FUNCTION_BLOCK FB_BMS
VAR PERSISTENT
	ui_CycleCount				: UINT;
	r_CumDischargeEnergy		: REAL; // kWh
	r_CumChargeEnergy			: REAL; // kWh
	r_maxVoltageEver	 		: REAL;
	r_maxChargeCurrentEver		: REAL;
	r_maxDischargeCurrentEver	: REAL;
	dt_LastCalibrationDate		: DT;
END_VAR

VAR_IN_OUT CONSTANT
	st_params	: st_BMS_Params;
END_VAR

VAR_IN_OUT
 	st_service	: st_BMS_service;
END_VAR

VAR_OUTPUT
	PowerStatus: eHVDC_Powerstatus := 0;
END_VAR
VAR_INPUT
	Set 					: st_BMS_Set;
	b_HVDCEnable			: BOOL;
	by_NoOfStrings			: BYTE;
END_VAR

VAR_OUTPUT
	get						: st_BMS_Get;
	b_InternalHVDCAllowed	:	BOOL;
END_VAR

VAR	
	InitDone			:	Bool := false;
	b_HVDC_OnRq			: BOOL;	
	FBState					:	ePOUState;
	IO					:	FB_BMS_IO;
	InitTimeout			: 	TON := (PT:=T#3S);
	BMS_24V_StartupTimer : TON := (PT := TIME#2S0MS);
	
	DeviceIDcounter		: WORD;
	
	//SFC
	SFCInit				: BOOL := FALSE;
	SFCReset			: BOOL := FALSE;
	
	//Modbus
	b_MBComErrorActive	: 	BOOL 	:= FALSE;
	ComTimer			:	Ton := (PT := TIME#100MS);
	t_TimeOut			: 	TIME := T#500MS;
	
	ResetBMS	:	Bool; 
	b_BMSShutdownRequested: BOOL;
	
	BMSReadIntervalTimer	 : TON := (PT := TIME#1S0MS);
	
	b_ManualReset	:BOOL;
	BMSDataValid		:	Bool;
	
	arDatalogMBMU	: ARRAY [0..58] OF WORD;
	arDatalogSBMU	: ARRAY[0..3] OF ARRAY[0..55] OF WORD;
	ARDatalogEMS	: ARRAY [0..16] OF WORD;
	
	AutoSOCCalibrationRequired	:	Bool;
END_VAR

VAR CONSTANT
	e_ID 				: eObject_ID := eObject_ID.Battery;
END_VAR

BMSDatalogger(b_enable := InitDone);
(*
FB_BMS

Inputs
	Set.b_EnableBMS				:	BOOL;
		Start BMS SFC sequence and initializes BMS. False means full BMS powerdown, so no status logging.
		With HVDC enabled, setting this value to False has no effect. Only after HVDC powerdown this value is tested.
		
	Set.b_ClearFault				:	BOOL;
		Clear errors and warning in BMS system. Set to true to initiate reset. Value resets automatically to false.
	
	Set.b_HVDC_Required			: 	BOOL;
		Set by FB_internalPowersupply. True initiates and keeps HVDC on, False initiates and retains powerdown

Outputs
	BMSGET
		-Some general status info
		-BATTinfo	struct with main operation battery data
		-MBMU_Status 	struct with detailed MBMU data
		-SBMU			Struct with detailed data per SBMU
		-Events			Warnings & Errors as per Sunspec list.
*)

IF InitDone THEN
	//INIT step
	//b_MBComErrorActive := FALSE;
	
	//CALL methods/functions
	//Link MBMU data when appropriate
	GetBatteryInfo(in := get.MBMU.BatteryStatus, OUT:= get.BatteryInfo);
	
	IF st_params.b_EnableAutoCalibration THEN
		IF dt_LastCalibrationDate > gvl.dt_SystemDateTime OR 
			(dt_LastCalibrationDate + st_params.T_AutoCalibrationInterval) < gvl.dt_SystemDateTime THEN
			get.T_RemainingTimeToAutoCalibration := T#0S;
			AutoSOCCalibrationRequired := TRUE;
		ELSE
			AutoSOCCalibrationRequired := FALSE;
			get.T_RemainingTimeToAutoCalibration := (dt_LastCalibrationDate + st_params.T_AutoCalibrationInterval) - gvl.dt_SystemDateTime;
		END_IF
	ELSE
		AutoSOCCalibrationRequired := FALSE;
		get.T_RemainingTimeToAutoCalibration := ST_Params.t_AutoCalibrationInterval;
	END_IF

		
	

	//get.LastCalibrationTime := dt_LastCalibrationDate;
	
	IF get.BatteryInfo.r_SOC < st_params.r_InternalConditioningSoCMin OR get.BatteryInfo.ar_CellVoltage[eSubValues.Minimum] < 3 THEN
		b_InternalHVDCAllowed := FALSE;
	ELSE
		b_InternalHVDCAllowed := TRUE;
	END_IF
	
	IO();
	
	BMSReadIntervalTimer(in:= not BMSReadIntervalTimer.Q);
	
	//Reset ErrorActive before entering SFC. 
	//any remaining error in the Modbus methods will set Erroractive again. 
	//This is pushed to events in BMS_Diagnostics
	
	//TEMPBMSHB();
	//hv required not allowed if BMS not enabled
	IF set.b_enable AND FBstate <> epoustate.EMSTOP THEN
		b_HVDC_OnRq := b_HVDCEnable OR st_params.b_forcePrecharging;
		
	ELSE
		b_HVDC_OnRq := FALSE;	
	END_IF
	
	//shutdown allowed if hvdc is offline
	b_BMSShutdownRequested := (NOT Set.b_Enable) AND get.MBMU.BatteryStatus.e_BMS_PowerOnStatus <> ePowerOnStatus.On; 
	
	IF b_ManualReset THEN
		Reset();
	END_IF
	
	//SFC delayed pulse trigger
	BMSSFC();
	
	BMS_Diagnostics();
	
	BMSDataValid := ((NOT get.Events.b_COMMUNICATION_ERROR) AND NOT (get.BatteryInfo.e_BMS_Status = eBMS_Status.Init));
END_IF

ACTION aBMSPoweroff:
IO.b_BMSEnable := FALSE;

get.BatteryInfo.b_BMSHeartBeatOK := FALSE;
get.BatteryInfo.e_BMS_PowerOnStatus := ePowerOnStatus.Off;
get.BatteryInfo.e_BMS_Status := eBMS_Status.Off;

get.MBMU.BatteryStatus.b_BMSHeartBeatOK := FALSE;
get.MBMU.BatteryStatus.e_BMS_PowerOnStatus := ePowerOnStatus.Off;
get.MBMU.BatteryStatus.e_BMS_Status := eBMS_Status.Off;

FBState := ePOUState.OFF;
END_ACTION

ACTION aBMSPowerOn:

//230V inverter requires some startup time. Start this first to init SBMU before MBMU
//This may not be needed, but the idea is to make sure the MBMU can reach the SBMU's at boot.
FBState := ePOUState.PowerUp;
io.b_BMSEnable := TRUE;
BMS_24V_StartupTimer(IN:=io.b_BMSEnable);
END_ACTION

ACTION aClearFaults:
SFCTip := ClearBMSFaults(st_params);
END_ACTION

ACTION aDisableInsulationMonitor:
SFCTip := OpenInsulationSwitch(st_params, TRUE);
END_ACTION

ACTION aGetMBMUData:
SFCTip := GetMBMUData(st_params);
END_ACTION

ACTION aGetSBMUData:
SFCTip := GetSBMUData(st_params);
END_ACTION

ACTION aGetStaticData:

IF (DeviceIDcounter=0) THEN
	IF GetMBMUStaticSystemData(st_params) THEN
		DeviceIDcounter:=1;
	END_IF;
ELSE
	IF GetSBMUStaticSystemData(st_params, DeviceIDcounter) THEN
		DeviceIDcounter := DeviceIDcounter+1;
	END_IF
	
	IF DeviceIDcounter > by_NoOfStrings THEN//BMSGet.MBMU_Status.by_NumberOfSubSystems THEN
		DeviceIDcounter:=0;
		SFCtip := NOT SFCtip;
	END_IF
END_IF
END_ACTION

ACTION aGetStatus:
IF GetSystemStatus(st_params) THEN
	IF FBState = ePOUState.PowerUp THEN FBState := ePOUState.Init; END_IF
	SFCtip := NOT SFCtip;
END_IF
END_ACTION

ACTION aInit:
DeviceIDcounter := 0;
SFCReset := FALSE;
b_MBComErrorActive := FALSE;
END_ACTION

ACTION aSetDateTime:
SFCTip := SetBMSDateTime(st_params);
END_ACTION

ACTION aSetPowerMode:
SFCTip := SetPowerMode(st_params);
END_ACTION

ACTION aWatchdog:
IF FBState = ePOUState.Init THEN FBState := ePOUState.Normal; END_IF

SFCtip := BMSHeartBeat(st_params);
DeviceIDcounter := 0;
END_ACTION

METHOD PRIVATE BMS_Diagnostics : BOOL
VAR
	
END_VAR

get.Events.b_COMMUNICATION_ERROR				:=	get.MBMU.GeneralSBMUStatus[6].5 	//SBMU CCAN comm lost
												OR get.MBMU.GeneralSBMUStatus[6].6 	//SBMU SCAN comm lost
												OR get.MBMU.GeneralSBMUStatus[6].7	//SBMU MCAN comm lost
												OR get.MBMU.MBMUStatus[0].6			//MBMU MCAN comm warning
												OR get.MBMU.MBMUStatus[0].7			//MBMU MCAN comm Lost
												OR get.MBMU.MBMUStatus[0].8			//SBMU EMS COMM lost
												OR get.MBMU.MBMUStatus[3].4			//SBMU MBMU comm fault
												OR b_MBComErrorActive;					//One or more Modbus communication errors 
									
get.Events.b_OVER_TEMP_ALARM					:= get.MBMU.GeneralSBMUStatus[2].1;	//single cell Overtemperature warning 4

get.Events.b_OVER_TEMP_WARNING				:= get.MBMU.GeneralSBMUStatus[1].14	//single cell Overtemperature warning 1
												OR get.MBMU.GeneralSBMUStatus[2].0; 	//single cell Overtemperature warning 2

get.Events.b_UNDER_TEMP_ALARM				:= FALSE; //no data

get.Events.b_UNDER_TEMP_WARNING				:= get.MBMU.GeneralSBMUStatus[2].2	//single cell Undertemperature warning 1
												OR get.MBMU.GeneralSBMUStatus[2].3 	//single cell Undertemperature warning 2
												OR get.MBMU.GeneralSBMUStatus[2].4; 	//single cell Undertemperature warning 3

get.Events.b_OVER_CHARGE_CURRENT_ALARM		:= get.MBMU.GeneralSBMUStatus[1].9;	//Charge Overcurrent warning 4

get.Events.b_OVER_CHARGE_CURRENT_WARNING		:= get.MBMU.GeneralSBMUStatus[1].6	//Charge Overcurrent warning 1
												OR get.MBMU.GeneralSBMUStatus[1].7 	//Charge Overcurrent warning 2
												OR get.MBMU.GeneralSBMUStatus[1].8; 	//Charge Overcurrent warning 3
											
get.Events.b_OVER_DISCHARGE_CURRENT_ALARM	:= get.MBMU.GeneralSBMUStatus[1].5;	//Discharge Overcurrent warning 4

get.Events.b_OVER_DISCHARGE_CURRENT_WARNING	:= get.MBMU.GeneralSBMUStatus[1].2	//Discharge Overcurrent warning 1
												OR get.MBMU.GeneralSBMUStatus[1].3 	//Discharge Overcurrent warning 2
												OR get.MBMU.GeneralSBMUStatus[1].4; 	//Discharge Overcurrent warning 3
											
get.Events.b_OVER_VOLT_ALARM					:= get.MBMU.GeneralSBMUStatus[0].6;	//Single cell extreme overVoltage warning

get.Events.b_OVER_VOLT_WARNING				:= get.MBMU.GeneralSBMUStatus[0].0	//Single cell overVoltage warning 1
												OR get.MBMU.GeneralSBMUStatus[0].1 	//Single cell overVoltage warning 2
												OR get.MBMU.GeneralSBMUStatus[0].2 	//Single cell overVoltage warning 3
												OR get.MBMU.GeneralSBMUStatus[0].8 	//Single rack overVoltage warning 1
												OR get.MBMU.GeneralSBMUStatus[0].9; 	//Single rack overVoltage warning 2
												
get.Events.b_UNDER_VOLT_ALARM				:= get.MBMU.GeneralSBMUStatus[0].7;	//Single cell extreme underVoltage warning

get.Events.b_UNDER_VOLT_WARNING				:= get.MBMU.GeneralSBMUStatus[0].3	//Single cell underVoltage warning 1
												OR get.MBMU.GeneralSBMUStatus[0].4 	//Single cell underVoltage warning 2
												OR get.MBMU.GeneralSBMUStatus[0].5 	//Single cell underVoltage warning 3
												OR get.MBMU.GeneralSBMUStatus[0].10 	//Single rack underVoltage warning 1
												OR get.MBMU.GeneralSBMUStatus[0].11; //Single rack underVoltage warning 2
												
get.Events.b_UNDER_SOC_MIN_ALARM				:= get.MBMU.GeneralSBMUStatus[6].14;	//r_SOC low warning 2

get.Events.b_UNDER_SOC_MIN_WARNING			:= get.MBMU.GeneralSBMUStatus[6].13;	//r_SOC low warning 1

get.Events.b_OVER_SOC_MAX_ALARM				:= FALSE; //no data

get.Events.b_OVER_SOC_MAX_WARNING			:= FALSE; //no data

get.Events.b_VOLTAGE_IMBALANCE_WARNING		:= get.MBMU.GeneralSBMUStatus[0].12;	//large voltage difference warning

get.Events.b_TEMPERATURE_IMBALANCE_ALARM		:= FALSE; //no data
												
get.Events.b_TEMPERATURE_IMBALANCE_WARNING	:= get.MBMU.GeneralSBMUStatus[2].5	//Large temperature difference warning 1
												OR get.MBMU.GeneralSBMUStatus[2].6 	//Large temperature difference warning 2
												OR get.MBMU.GeneralSBMUStatus[2].7; 	//Large temperature difference warning 3
												
get.Events.b_CONTACTOR_ERROR					:= get.MBMU.GeneralSBMUStatus[5].1	//Main positive relay sticking
												OR get.MBMU.GeneralSBMUStatus[5].2 	//Main negative relay sticking
												OR get.MBMU.GeneralSBMUStatus[5].3 	//Both main relays sticking
												OR get.MBMU.GeneralSBMUStatus[5].4 	//Main positive relay open
												OR get.MBMU.GeneralSBMUStatus[5].5 	//Main negative relay open
												OR get.MBMU.GeneralSBMUStatus[6].15; //HV open circuit warning
												
get.Events.b_FAN_ERROR						:= get.MBMU.GeneralSBMUStatus[5].7;	//main control box fan warning

get.Events.b_GROUND_FAULT					:= FALSE; //no data

get.Events.b_OPEN_DOOR_ERROR					:= FALSE; //no data

get.Events.b_CURRENT_IMBALANCE_WARNING		:= FALSE; //no data

get.Events.b_OTHER_ALARM						:= get.MBMU.GeneralSBMUStatus[0].13	//Invalid voltage warning
												OR get.MBMU.GeneralSBMUStatus[1].10 	//Current sensor fault
												OR get.MBMU.GeneralSBMUStatus[2].15 //single temperature sampling abnormal value warning
												OR get.MBMU.GeneralSBMUStatus[3].0 	//multiple temperature sampling abnormal value warning
												OR get.MBMU.GeneralSBMUStatus[4].9 	//CSC supply abnormal
												OR get.MBMU.GeneralSBMUStatus[4].10 	//SBMU supply abnormal
												OR get.MBMU.GeneralSBMUStatus[4].14 	//MSD warning
												OR get.MBMU.GeneralSBMUStatus[4].15 	//rack fuse warning
												OR get.MBMU.GeneralSBMUStatus[6].11 	//cell balance circuit short
												OR get.MBMU.GeneralSBMUStatus[7].3 	//precharching failed twice
												OR get.MBMU.MBMUStatus[1].7 			//estop fault
												OR get.MBMU.MBMUStatus[3].3; 		//MBMU 24V fault
												
get.Events.b_OTHER_WARNING					:= get.MBMU.MBMUStatus[0].0 			//insulation warning
												OR get.MBMU.MBMUStatus[1].10 		//rack fan warning
												OR get.MBMU.MBMUStatus[3].7;			//TMS warning

get.Events.b_DISCONNECTOR_OFF				:= get.MBMU.GeneralSBMUStatus[5].0;	//rack isolate switch warning		
					
get.Events.b_CONFIGURATION_ALARM				:= get.MBMU.GeneralSBMUStatus[5].6 	//battery rack door fault
												OR get.MBMU.GeneralSBMUStatus[5].9 	//rack fire system level 1 fault
												OR get.MBMU.GeneralSBMUStatus[5].10 	//smoke detector contact open
												OR get.MBMU.GeneralSBMUStatus[5].11 	//temp detector contact open
												OR get.MBMU.GeneralSBMUStatus[5].14 	//aerosol warning
												OR get.MBMU.GeneralSBMUStatus[6].0 	//rack fire system level 2 fault
												OR get.MBMU.GeneralSBMUStatus[6].10 	//SBMU TMS CCAN comm lost with hv on
												OR get.MBMU.GeneralSBMUStatus[7].0 	//lvl 3 fault tms
												OR get.MBMU.GeneralSBMUStatus[7].1 	//TMS mode conflict
												OR get.MBMU.GeneralSBMUStatus[7].2 	//TMS warning
												OR get.MBMU.GeneralSBMUStatus[8].0 	//Thermal runaway caused fire
												OR get.MBMU.MBMUStatus[0].1	 		//Insulation fault
												OR get.MBMU.MBMUStatus[0].2			//Insulation error
												OR get.MBMU.MBMUStatus[0].3 			//Less HV racks than expected
												OR get.MBMU.MBMUStatus[0].9			//IMM comm fault
												OR get.MBMU.MBMUStatus[0].10 		//Air conditioning comm fault
												OR get.MBMU.MBMUStatus[0].11			//TMS comm fault
												OR get.MBMU.MBMUStatus[0].13			//TMS comm fault lvl 2
												OR get.MBMU.MBMUStatus[0].14 		//TMS mode conflict
												OR get.MBMU.MBMUStatus[0].15			//TMS comm fault level 1
												OR get.MBMU.MBMUStatus[1].3	 		//AUX power DCDC failure
												OR get.MBMU.MBMUStatus[1].4			//Fire system fault lvl 1
												OR get.MBMU.MBMUStatus[1].5 			//Fire system fault lvl 2
												OR get.MBMU.MBMUStatus[1].6			//Fire system failure warning
												OR get.MBMU.MBMUStatus[1].8	 		//client estop fault
												OR get.MBMU.MBMUStatus[1].9			//rack door fault
												OR get.MBMU.MBMUStatus[1].12;		//smoke ex fan body fault
								
get.Events.b_CONFIGURATION_WARNING			:= get.MBMU.GeneralSBMUStatus[6].8	//SBMU TMS CCAN comm lost
												OR get.MBMU.MBMUStatus[0].12	 		//TMS comm warning
												OR get.MBMU.MBMUStatus[1].0			//SPD failure
												OR get.MBMU.MBMUStatus[1].1 			//Aux power DCDC failure
												OR get.MBMU.MBMUStatus[1].2			//AUX power DCDC failure
												OR get.MBMU.MBMUStatus[1].6 			//Fire system failure warning
												OR get.MBMU.MBMUStatus[1].11;		//Smoke exhaust fan body warning

get.Events.b_POWERONFAULT					:= get.MBMU.BatteryStatus.e_BMS_PowerOnStatus = ePoweronstatus.PowerOn_Fault;
get.Events.b_Powerofffault					:= get.MBMU.BatteryStatus.e_BMS_PowerOnStatus = ePoweronstatus.PowerOff_Fault;
END_METHOD

METHOD BMSDatalogger : BOOL
VAR_INPUT
	b_enable	: BOOL;
END_VAR

VAR_INST
	LogTimer 	: TON := (PT := T#15S);
	ArrayCounter	:	UINT := 0;
	SBMUCounter		:	UINT	:=	0;
	LogStep			:	UINT := 0;	

	s_MBMUData	:	STRING(255);
	s_SBMUData	:	ARRAY[0..3] OF STRING (255);
	s_EMSData	:	STRING(255);
END_VAR
LogTimer(in := NOT LogTimer.Q);	//start data logging at interval

CASE logstep OF
	0:	//do nothing
		IF LogTimer.Q THEN
			LogStep	:=	1;
		END_IF
		
	1:	//Write MBMU data
		s_MBMUData := '';
		FOR ArrayCounter := 0 TO 52 DO
			s_MBMUData := Concat(s_MBMUData, Word_to_hexstr(arDatalogMBMU[ArrayCounter], 2, FALSE));
		END_FOR
		Logstep := 2;
		
	2: //Write data of 1 SMBU //required log frequency is lower, so send each separate to save data and cpu load 
		s_SBMUData[SBMUCounter] := '';
		FOR ArrayCounter := 0 TO 50 DO
			s_SBMUData[SBMUCounter] := Concat(s_SBMUData[SBMUCounter], Word_to_hexstr(arDatalogSBMU[SBMUCounter][ArrayCounter], 2, FALSE));
		END_FOR
		
		SBMUCounter := SBMUCounter+1;
		IF SBMUCounter >= by_NoOfStrings THEN
			SBMUCounter := 0;
			Logstep := 3;
		END_IF

	3: //Write data of EMS
		s_EMSData := '';
		FOR ArrayCounter := 0 TO 5 DO
			s_EMSData := Concat(s_EMSData, Word_to_hexstr(arDatalogEMS[ArrayCounter], 2, FALSE));
		END_FOR	
		Logstep := 0;
END_CASE

MQTTComOpenremote.FillBatteryDatalog(s_MBMUData := s_MBMUData, s_SBMUData := s_SBMUData, s_EMSData := s_EMSData);
END_METHOD

METHOD PRIVATE BMSHeartBeat : BOOL

VAR_IN_OUT CONSTANT
	st_params			: ST_BMS_params;
END_VAR

VAR_INST
	WriteReg		:	FB_MBWriteSingleReg;
	ReadReg			:	FB_MBReadRegs;
	
	readbCommBusy		:	BOOL;
	readbComError		:	BOOL;
	readerrID			:	UDINT;
	
	WritebCommBusy		:	BOOL;
	WritebComError		:	BOOL;
	WriteerrID			:	UDINT;
	
	ReadDone			:	F_Trig;
	ReadOK				: 	BOOL;
	WriteDone			:	F_Trig;
	WriteOK				: 	BOOL;
	
	//ComTimer		:	Ton := (PT := TIME#0S200MS);
	
	OldValue		:	WORD := 0;
	BMSHBValue		:	WORD := 0;
	
	WatchdogUpdateTimer	:	Tof := (PT := TIME#3S0MS);
	WatchdogCommTimer	:	Tof := (PT := TIME#3S0MS);
	
	ComRetryCounter	:	USINT := 0;
END_VAR
ComTimer(in := NOT(ComTimer.Q OR readbCommBusy OR WritebCommBusy));

ReadReg(
sIPAddr := st_params.IP_BMS,
nTCPPort := 502,
nUnitID := 255,//16#FF;
nMBAddr := 768,
nQuantity := 1,
cbLength := 2,
pDestAddr := ADR(BMSHBValue),
bExecute := ComTimer.Q,
tTimeOut := t_TimeOut,
bBusy => readbCommBusy,
bError => readbComError,
nErrId => readerrID,
cbRead => 
);

ReadDone(clk := readbCommBusy);
ReadOK := ReadDone.Q AND NOT readbComError;

//read value is transmitted back into the write buffer if read is succesful
//BMS increments this value every second.
WriteReg(
sIPAddr := st_params.IP_BMS,
nTCPPort := 502,
nUnitID := 255,//16#FF;
nMBAddr := 896,
nValue := BMSHBValue,
tTimeout := T#1000MS,
bExecute := ReadOK,
bBusy => WritebCommBusy,
bError => WritebComError,
nErrId => WriteerrID,
);

WriteDone(clk := writebCommBusy);
WriteOK := writeDone.Q AND NOT writebComError;

//if written value and BMS value are equal for longer than 3 seconds, the BMS isn't incrementing the value anymore or communication failed.
//BMS itself will throw warning after 30s and disable 10s after that.
WatchdogUpdateTimer(in:= (OldValue <> BMSHBValue));
OldValue := BMSHBValue;

//if modbus communication throws an error retry for 3s, otherwise system failed.
//WatchdogCommTimer(in:= WriteOK);

//both values are normally high and fall away if they timeout
get.BatteryInfo.b_BMSHeartBeatOK := WatchdogUpdateTimer.Q;// OR WatchdogCommTimer.Q;
get.MBMU.BatteryStatus.b_BMSHeartBeatOK := WatchdogUpdateTimer.Q;

IF (ReadDone.Q AND readbComError) OR (WriteDone.Q AND WritebComError) THEN
	ComRetryCounter := ComRetryCounter + 1;
	IF COMRetryCounter > 5 THEN
		b_MBComErrorActive := TRUE;
		get.BatteryInfo.b_BMSHeartBeatOK := FALSE;
	END_IF
END_IF

IF ReadOK THEN
	arDatalogMBMU[47] := BMSHBValue;
END_IF

IF WriteOK THEN
	arDatalogEMS[0] := BMSHBValue;
	ComRetryCounter := 0;
	BMSHeartBeat := TRUE;
	b_MBComErrorActive := FALSE;
END_IF
END_METHOD

ACTION BMSSFC:
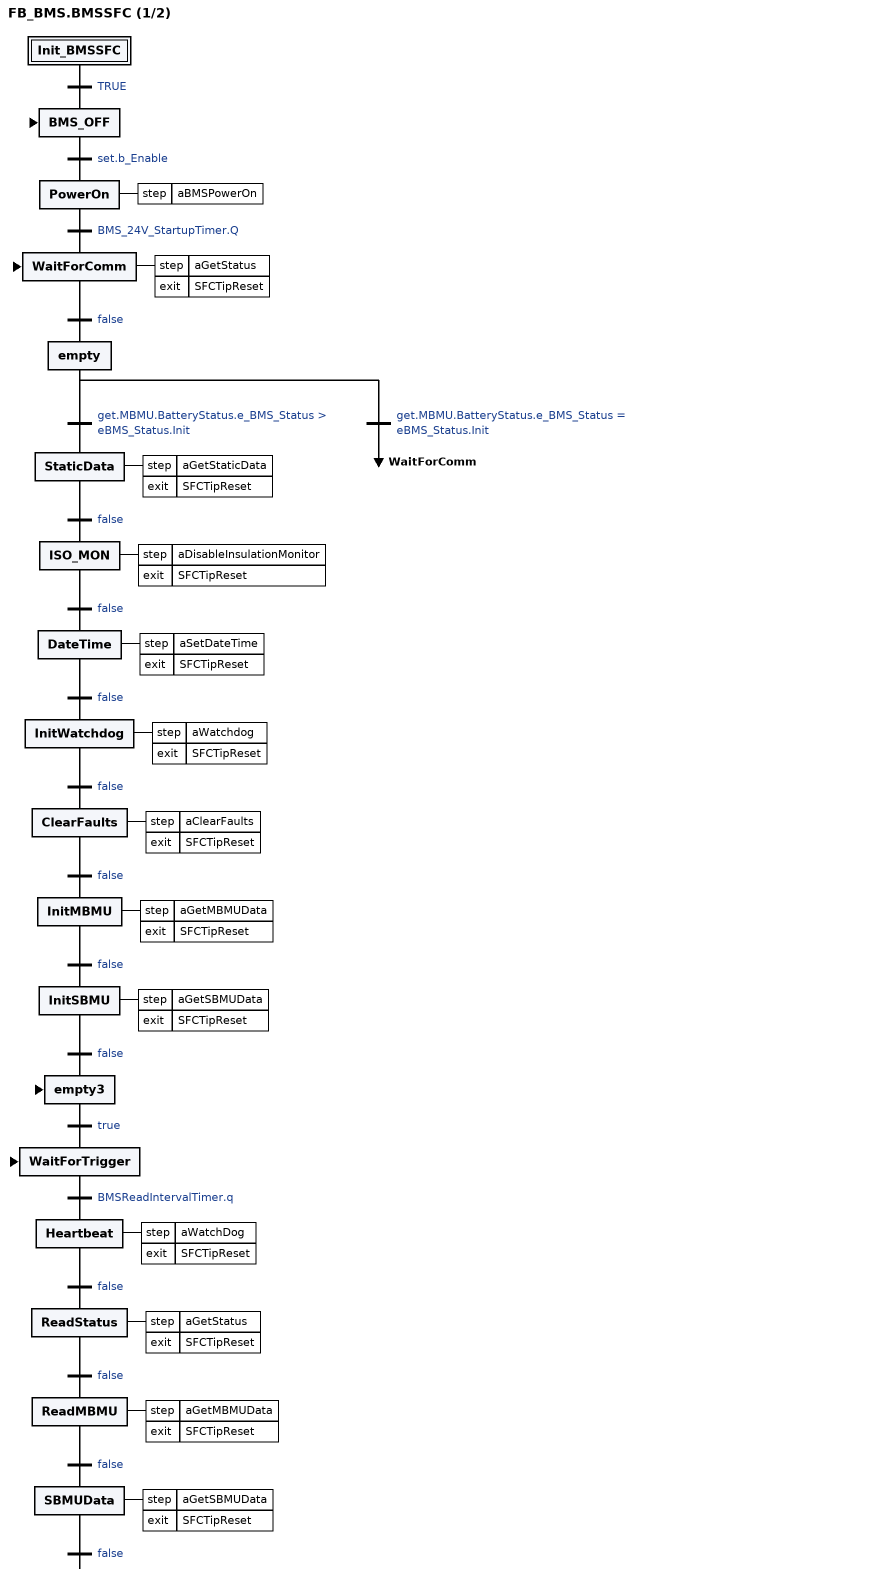
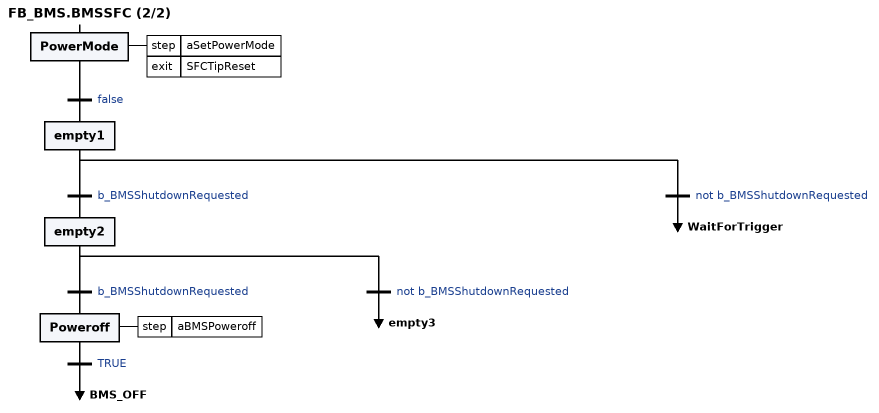
INITIAL_STEP Init_BMSSFC:
END_STEP
TRANSITION FROM Init_BMSSFC TO BMS_OFF
    := TRUE;
END_TRANSITION
STEP BMS_OFF:
END_STEP
TRANSITION FROM BMS_OFF TO PowerOn
    := set.b_Enable;
END_TRANSITION
// macro BMSInit begins
STEP PowerOn:
    aBMSPowerOn(N);  // step action
END_STEP
TRANSITION FROM PowerOn TO WaitForComm
    := BMS_24V_StartupTimer.Q;
END_TRANSITION
STEP WaitForComm:
    aGetStatus(N);  // step action
    SFCTipReset(P0);  // exit action
END_STEP
TRANSITION FROM WaitForComm TO empty
    := false;
END_TRANSITION
STEP empty:
END_STEP
TRANSITION FROM empty TO StaticData
    := get.MBMU.BatteryStatus.e_BMS_Status > eBMS_Status.Init;
END_TRANSITION
TRANSITION FROM empty TO WaitForComm
    := get.MBMU.BatteryStatus.e_BMS_Status = eBMS_Status.Init;
END_TRANSITION
STEP StaticData:
    aGetStaticData(N);  // step action
    SFCTipReset(P0);  // exit action
END_STEP
TRANSITION FROM StaticData TO ISO_MON
    := false;
END_TRANSITION
STEP ISO_MON:
    aDisableInsulationMonitor(N);  // step action
    SFCTipReset(P0);  // exit action
END_STEP
TRANSITION FROM ISO_MON TO DateTime
    := false;
END_TRANSITION
STEP DateTime:
    aSetDateTime(N);  // step action
    SFCTipReset(P0);  // exit action
END_STEP
TRANSITION FROM DateTime TO InitWatchdog
    := false;
END_TRANSITION
STEP InitWatchdog:
    aWatchdog(N);  // step action
    SFCTipReset(P0);  // exit action
END_STEP
TRANSITION FROM InitWatchdog TO ClearFaults
    := false;
END_TRANSITION
STEP ClearFaults:
    aClearFaults(N);  // step action
    SFCTipReset(P0);  // exit action
END_STEP
TRANSITION FROM ClearFaults TO InitMBMU
    := false;
END_TRANSITION
STEP InitMBMU:
    aGetMBMUData(N);  // step action
    SFCTipReset(P0);  // exit action
END_STEP
TRANSITION FROM InitMBMU TO InitSBMU
    := false;
END_TRANSITION
STEP InitSBMU:
    aGetSBMUData(N);  // step action
    SFCTipReset(P0);  // exit action
END_STEP
TRANSITION FROM InitSBMU TO empty3
    := false;
END_TRANSITION
STEP empty3:
END_STEP
TRANSITION FROM empty3 TO WaitForTrigger
    := true;
END_TRANSITION
// macro BMSActive begins
STEP WaitForTrigger:
END_STEP
TRANSITION FROM WaitForTrigger TO Heartbeat
    := BMSReadIntervalTimer.q;
END_TRANSITION
STEP Heartbeat:
    aWatchDog(N);  // step action
    SFCTipReset(P0);  // exit action
END_STEP
TRANSITION FROM Heartbeat TO ReadStatus
    := false;
END_TRANSITION
STEP ReadStatus:
    aGetStatus(N);  // step action
    SFCTipReset(P0);  // exit action
END_STEP
TRANSITION FROM ReadStatus TO ReadMBMU
    := false;
END_TRANSITION
STEP ReadMBMU:
    aGetMBMUData(N);  // step action
    SFCTipReset(P0);  // exit action
END_STEP
TRANSITION FROM ReadMBMU TO SBMUData
    := false;
END_TRANSITION
STEP SBMUData:
    aGetSBMUData(N);  // step action
    SFCTipReset(P0);  // exit action
END_STEP
TRANSITION FROM SBMUData TO PowerMode
    := false;
END_TRANSITION
STEP PowerMode:
    aSetPowerMode(N);  // step action
    SFCTipReset(P0);  // exit action
END_STEP
TRANSITION FROM PowerMode TO empty1
    := false;
END_TRANSITION
STEP empty1:
END_STEP
TRANSITION FROM empty1 TO empty2
    := b_BMSShutdownRequested;
END_TRANSITION
TRANSITION FROM empty1 TO WaitForTrigger
    := not b_BMSShutdownRequested;
END_TRANSITION
STEP empty2:
END_STEP
TRANSITION FROM empty2 TO Poweroff
    := b_BMSShutdownRequested;
END_TRANSITION
TRANSITION FROM empty2 TO empty3
    := not b_BMSShutdownRequested;
END_TRANSITION
STEP Poweroff:
    aBMSPoweroff(N);  // step action
END_STEP
TRANSITION FROM Poweroff TO BMS_OFF
    := TRUE;
END_TRANSITION
// branch label Branch1_BMSSFC
// branch label Branch0_BMSSFC
END_ACTION

METHOD PRIVATE CalculateCumulativeValues
VAR_IN_OUT
	get : st_BMS_BatterySummary;
END_VAR

VAR_INPUT
	t_cycletime			: TIME;
END_VAR

VAR
	timefraction		: REAL;
	millisInHour		: REAL := 3600000;
	ui_cyclecountTemp : UINT;
END_VAR

VAR_INST
	r_trigResetCounters		: r_trig;
	ton_EnergyPulseTimer	: TON := (PT:= T#10MS);
END_VAR
timefraction := TO_REAL(t_cycletime) / millisInHour;

IF get.r_SystemPower > 0 THEN
	get.r_HistAccDischargeEnergy := get.r_HistAccDischargeEnergy + ABS(get.r_SystemPower) * timefraction;
ELSIF get.r_SystemPower < 0 THEN
	get.r_HistAccChargeEnergy := get.r_HistAccDischargeEnergy + ABS(get.r_SystemPower) * timefraction;
END_IF

//Get current cycle count
get.ui_CycleCount := TO_UINT(get.r_HistAccDischargeEnergy / MAX(1, get.r_ratedEnergyCapacity));



//--- store max charge/discharge current to persistent var ---
IF get.r_SystemCurrent > 0 AND get.r_SystemCurrent > r_maxDischargeCurrentEver THEN
	r_maxDischargeCurrentEver := get.r_SystemCurrent;
ELSIF get.r_SystemCurrent < 0 AND ABS(get.r_SystemCurrent) > r_maxChargeCurrentEver THEN
	r_maxChargeCurrentEver := ABS(get.r_SystemCurrent);
END_IF
//overwrite to original structure
get.r_maxDischargeCurrentEver := r_maxDisChargeCurrentEver;
get.r_maxChargeCurrentEver := r_maxChargeCurrentEver;

//--- store max voltage to persistent var ---
IF get.r_SystemVoltage > 0 AND get.r_Systemvoltage > r_maxVoltageEver THEN
	r_maxVoltageEver := get.r_SystemVoltage;
END_IF
//overwrite to original structure
get.r_maxVoltageEver := r_maxVoltageEver;

r_trigResetCounters(CLK:= st_params.b_ResetPersistentVars);
IF r_trigResetCounters.Q THEN
	r_maxVoltageEver := 0;
	r_maxChargeCurrentEver := 0;
	r_maxDisChargeCurrentEver := 0;
END_IF
END_METHOD

METHOD PRIVATE CalculatedRatings : BOOL
VAR_INPUT
	numberofstrings : BYTE;
END_VAR
get.BatteryInfo.r_ratedEnergyCapacity := st_params.r_kWhperString * numberofstrings;

IF get.BatteryInfo.r_ratedEnergyCapacity <> 0 THEN
	get.BatteryInfo.r_ratedCurrent := st_params.r_CrateBattery * st_params.r_AhperString * numberofstrings;
	get.BatteryInfo.r_ratedPower := st_params.r_CrateBattery * get.BatteryInfo.r_ratedEnergyCapacity;
END_IF
END_METHOD

METHOD PRIVATE CalculateSoCUser : BOOL
VAR_IN_OUT
	get : ST_BMS_get;
	set	: ST_BMS_Set;
END_VAR

VAR_IN_OUT CONSTANT
	st_params	: st_BMS_Params;
END_VAR

VAR_INST
	r_Soc							: REAL;
	fb_SOCLowLimit					: fbValueOutOfRange;
	fb_SOCHighLimit					: fbValueOutOfRange;
	r_SoCMinActual 					: REAL;
	r_SoCMaxActual					: REAL;
	r_deltaSoC						: REAL;
	r_ratio							: REAL;
	r_offset						: REAL;
	
	RS_chargingAllowed				: RS;
	RS_DischargingAllowed			: RS;
END_VAR
//Calculations
r_deltaSoC:= st_params.r_SoCAbsoluteMax - st_params.r_SoCAbsoluteMin;
r_ratio := 1 / SEL(r_deltaSoC=0,r_deltaSoC/100,1);
r_offset := st_params.r_SoCAbsoluteMin * r_Ratio;


//user soc setpoint, first limit user value with 100% and scale to original battery soc 
r_SoCMinActual := (LIMIT(0, set.r_SocMin, set.r_SocMax) + r_Offset) / r_ratio;
r_SoCMaxActual := sel(AutoSOCCalibrationRequired,(LIMIT(set.r_SocMin,set.r_SocMax,100) + r_Offset) / r_ratio, 100);

//Set limit with error when hard limits exceed absolute VDL limits
fb_SOCLowLimit(
	r_var		:= r_SocMinActual, 
	r_min		:= st_params.r_SoCAbsoluteMin, 
	r_max		:= st_params.r_SoCAbsoluteMax,
	r_WhenError := st_params.r_SoCAbsoluteMin,
	b_IsError	=> get.events.b_SoCLowLimitOutOfRange);

fb_SOCHighLimit(
	r_var		:= r_SocMaxActual, 
	r_min		:= st_params.r_SoCAbsoluteMin, 
	r_max		:= st_params.r_SoCAbsoluteMax,
	r_WhenError := st_params.r_SoCAbsoluteMin,
	b_IsError	=> get.events.b_SoCHighLimitOutOfRange);


//Set scaled soc to monitoring
get.BatteryInfo.r_SOCScaled := F_RoundReal(LIMIT(0, get.BatteryInfo.r_SOC * r_ratio - r_offset, 100),1); // set limit to avoid exceed 0 or 100%.

//set scaled kwh discharging remaining
get.BatteryInfo.r_RemainingDischargeEnergyNett := r_deltaSoC/ 100 * get.BatteryInfo.r_RemainingDischargeEnergy;
get.BatteryInfo.r_RemainingChargeEnergyNett := r_deltaSoC/ 100 * get.BatteryInfo.r_RemainingChargeEnergy;

r_Soc := get.BatteryInfo.r_SoC;
//Set Charge only when soft high limit reached
rs_dischargingAllowed(
	set:=r_SoC > (r_SoCMinActual + st_params.r_SocHysteresis),
	Reset1 := r_SoC <= r_SoCMinActual OR get.BatteryInfo.e_BMS_Status = eBMS_Status.FullDischarge,
	Q1 => get.BatteryInfo.b_dischargingAllowed);

//Set discharge only when soft high limit reached
rs_chargingAllowed(
	SET:= r_SoC < (r_SoCMaxActual - st_params.r_SocHysteresis),
	RESET1:= r_SoC >= r_SoCMaxActual OR get.BatteryInfo.e_BMS_Status = eBMS_Status.FullCharge,
	Q1=> get.BatteryInfo.b_chargingAllowed);
END_METHOD

METHOD PRIVATE CalculateTimeRemaining : BOOL
VAR_INPUT
END_VAR

VAR_OUTPUT
END_VAR

VAR_INST
	a_PowerArray			: ARRAY [1..20] OF REAL;
	st_Params_MA			: ST_CTRL_MOVING_AVERAGE_PARAMS;
	ui_filterSize			: UINT := 10;
	fb_SmoothPower			: FB_CTRL_MOVING_AVERAGE;
	r_PowerMA				: REAL;
	r_HoursRemaining		: REAL;
END_VAR
//SMOOTH SETPOINT VALUE SINCE VALUE IS SWITCHED RAPIDLY BETWEEN UPPER AND LOWER GRID LIMIT.
st_Params_MA.tCtrlCycleTime := T#100MS;
	st_Params_MA.tTaskCycleTime := T#1MS;
	st_Params_MA.nWorkArray_SIZEOF := SIZEOF(a_PowerArray);
	st_Params_MA.pWorkArray_ADR	:= ADR(a_PowerArray);
	st_Params_MA.nSamplesToFilter:= ui_filterSize;

fb_SmoothPower(fin:= get.BatteryInfo.r_SystemPower,
				eMode := E_CTRL_MODE.eCTRL_MODE_ACTIVE,
				fout=> r_PowerMA,
				stParams := st_Params_MA);
				
r_HoursRemaining := get.BatteryInfo.r_RemainingDischargeEnergyNett / MAX(1, r_PowerMA);
END_METHOD

METHOD PRIVATE ClearBMSFaults : BOOL
VAR_IN_OUT CONSTANT
	st_params			: ST_BMS_params;
END_VAR

VAR_INST
	WriteRegSet		:	FB_MBWriteSingleReg;
	WriteRegClear	:	FB_MBWriteSingleReg;
	
	bCommBusy	:	BOOL;
	bComError	:	BOOL;
	errID		:	UDINT;
	b_ClearDone	:	BOOL := FALSE;

	w_ClearFault	:	WORD;
	TX1Done 	: 	f_trig;
	
	bCommBusy2	:	BOOL;
	bComError2	:	BOOL;
	errID2		:	UDINT;
	TX2Done 	: 	f_trig;

	ComRetryCounter	:	USINT := 0;	
	
	ResetDelayTimer	: Tp := (PT:=T#500MS);
END_VAR
//Catl says we need to write 1 to clear, then write back to 0 to be able to log new errors.
//This method is called continuously when bms is active. It will usually write zero's.
//If set.b_ClearFault is 1, that will be written. The value will be cleared by this method after the write so next write will be a 0 again.
//With this, a reset cycle takes half a second with the current ComTimer.

ClearBMSFaults := FALSE;

ComTimer(in := NOT(ComTimer.Q OR bCommBusy));

//first write clearing register to 1
WriteRegSet(
	sIPAddr := st_params.IP_BMS,
	nTCPPort := 502,
	nUnitID := 255,//16#FF;
	nMBAddr := 908,
	nValue := 1,
	tTimeOut := t_TimeOut,
	bExecute := ComTimer.Q,
	bBusy => bCommBusy,
	bError => bComError,
	nErrId => errID,
);

TX1Done(CLK := bCommBusy);
b_ClearDone	:= 	TX1Done.Q AND NOT bComError;
ResetDelayTimer(in:=b_ClearDone);
//reset value back to 0 afterwards. CATL requirement
WriteRegClear(
	sIPAddr := st_params.IP_BMS,
	nTCPPort := 502,
	nUnitID := 255,//16#FF;
	nMBAddr := 908,
	nValue := 0,
	tTimeout := T#100MS,
	bExecute := NOT ResetDelayTimer.Q,
	bBusy => bCommBusy2,
	bError => bComError2,
	nErrId => errID2
);

TX2Done(CLK := bCommBusy2);

IF (TX1Done.Q AND bComError) OR (TX2Done.Q AND bComError2) THEN
	ComRetryCounter := ComRetryCounter + 1;
	IF COMRetryCounter > 5 THEN
		b_MBComErrorActive := TRUE;
		ClearBMSFaults := TRUE;
	END_IF
END_IF

IF (TX1Done.Q AND NOT bComError) THEN
	arDatalogEMS[4] := 1;	
END_IF

IF TX2Done.Q AND NOT bComError2 THEN
	arDatalogEMS[4] := 0;	
	b_MBComErrorActive := FALSE;
	ComRetryCounter := 0;
	ClearBMSFaults := TRUE;
END_IF
END_METHOD

METHOD EMSTOP : BOOL
EMSTOP := FALSE;

FBState := ePOUState.EMSTOP;

IF get.MBMU.BatteryStatus.e_BMS_PowerOnStatus <> ePowerOnStatus.On THEN
	EMSTOP := TRUE;
END_IF
END_METHOD

METHOD PRIVATE GetBatteryInfo : BOOL

VAR_IN_OUT
	IN : ST_MBMU_BatterySummary;
	OUT: ST_BMS_BatterySummary;
END_VAR


VAR_INST
	ton_syncPulse : TON := (PT := T#100MS);
	t_SyncTimer	: TIME := T#100MS;
	tof_Release : TOF := (PT:= T#2S);
END_VAR
tof_Release(IN:= get.Events.b_COMMUNICATION_ERROR OR get.MBMU.BatteryStatus.r_SOC > 101);

//set batterysummery data if MBMU gives no shit.
IF ton_syncPulse.Q THEN
	IF NOT tof_Release.Q THEN
		//copy inherited data from original location.
 		MEMCPY(ADR(OUT), ADR(IN), SIZEOF(IN));
		//generate additional data
		CalculateSoCUser(get := get, set := set, st_params:=st_params);
		CalculatedRatings(numberOfStrings:= settings.Configuration.by_NoBatteryStrings);
		CalculateCumulativeValues(get := OUT, t_cycleTime := t_syncTimer);
	ELSE
		out.ar_CellTemperature[0] := -273;
		out.ar_CellTemperature[1] := -273;
		out.ar_CellTemperature[2] := -273;
	END_IF
END_IF
 

ton_syncPulse(IN := NOT ton_syncPulse.Q, PT := t_SyncTimer);
END_METHOD

METHOD PRIVATE GetCellData : BOOL
VAR_IN_OUT CONSTANT
	st_params			: ST_BMS_params;
END_VAR

VAR_INPUT
	SBMUID	:	BYTE;	//SBMU 1-#ofstrings
	CSCID	:	BYTE;	//CSC 1-4
END_VAR

VAR_OUTPUT
	CellVoltages		:	ARRAY[1..52] OF REAL;
	Celltemperatures	:	ARRAY[1..16] OF INT;
	BalanceStatus		:	ARRAY[1..4] OF WORD; //bit per cell?
END_VAR

VAR_INST
	MBReadCellVoltages	: 	FB_MBReadRegs;
	MBReadTemperatures	: 	FB_MBReadRegs;
	MBReadCellBalance	: 	FB_MBReadRegs;
	
//	CellVoltageData		: 	ARRAY[1..52] OF WORD;
	TemperatureData		: 	ARRAY[1..16] OF BYTE;
//	CellBalanceData		: 	ARRAY[1..4] OF WORD;
	
	bCommBusy			:	ARRAY[1..3] OF BOOL;
	bComError			:	ARRAY[1..3] OF BOOL;
	errID				:	ARRAY[1..3] OF UDINT;
	cbRead				:	ARRAY[1..3] OF UDINT;
	TransmissionDone	: 	ARRAY[1..3] OF f_trig;
	
	DataComplete		:	ARRAY[1..3] OF BOOL;
	
	//ComTimer			:	Ton := (PT := TIME#0S500MS);
END_VAR

VAR
	LoopCounter			:	INT;
END_VAR

GetCellData := FALSE;

IF (SBMUID < 1) OR (SBMUID > get.MBMU.by_NumberOfSubSystems) THEN
	GetCellData := TRUE;
	RETURN;
END_IF
IF (CSCID < 1) OR (CSCID > 4) THEN
	GetCellData := TRUE;
	RETURN;
END_IF

ComTimer(in := NOT(ComTimer.Q OR bCommBusy[1] OR bCommBusy[2] OR bCommBusy[3]));

IF ComTimer.Q THEN
	DataComplete[1] := FALSE;
	DataComplete[2] := FALSE;
	DataComplete[3] := FALSE;
END_IF

MBReadCellVoltages(
sIPAddr := st_params.IP_BMS,
nTCPPort := 502,
nUnitID := 255,//16#FF;
nMBAddr := (SBMUID*1024)+128+(52*(CSCID-1)),	//SBMU 1, module 1, start at 0x0480, increment 52 per module & 1024 per sbmu
nQuantity := 52,
cbLength := SIZEOF(CellVoltages),
pDestAddr := ADR(CellVoltages),
bExecute := ComTimer.Q,
bBusy => bCommBusy[1],
bError => bComError[1],
nErrId => errID[1],
cbRead => cbRead[1],
tTimeOut := t_TimeOut,
);

MBReadTemperatures(
sIPAddr := st_params.IP_BMS,
nTCPPort := 502,
nUnitID := 1,//16#FF;
nMBAddr := (SBMUID*1024)+704+(8*(CSCID-1)),	//SBMU 1, module 1, start at 0x06c0, increment 8 (16 byte) per module & 1024 per sbmu
nQuantity := 8*2,
cbLength := SIZEOF(TemperatureData),
pDestAddr := ADR(TemperatureData),
bExecute := ComTimer.Q,
bBusy => bCommBusy[2],
bError => bComError[2],
nErrId => errID[2],
cbRead => cbRead[2],
tTimeOut := t_TimeOut,
);

MBReadTemperatures(
sIPAddr := st_params.IP_BMS,
nTCPPort := 502,
nUnitID := 1,//16#FF;
nMBAddr := (SBMUID*1024)+912+(4*(CSCID-1)),	//SBMU 1, module 1, start at 0x0790, increment 4 per module & 1024 per sbmu
											//not sure if CSC2 starts at address 4, or immediatly follows after last cell of csc1.
nQuantity := 4*2,
cbLength := SIZEOF(BalanceStatus),
pDestAddr := ADR(BalanceStatus),
bExecute := ComTimer.Q,
bBusy => bCommBusy[3],
bError => bComError[3],
nErrId => errID[3],
cbRead => cbRead[3],
tTimeOut := t_TimeOut,
);

TransmissionDone[1](clk:=bCommBusy[1]);
TransmissionDone[2](clk:=bCommBusy[2]);
TransmissionDone[3](clk:=bCommBusy[3]);

IF TransmissionDone[1].Q AND NOT bComError[1] THEN
	DataComplete[1] := TRUE;
END_IF

IF TransmissionDone[2].Q AND NOT bComError[2] THEN
	FOR loopcounter := 1 TO 16 BY 1 DO
		Celltemperatures[loopcounter] := TemperatureData[loopcounter]-50;
	END_FOR
	DataComplete[2] := TRUE;
END_IF

IF TransmissionDone[1].Q AND NOT bComError[1] THEN
	DataComplete[3] := TRUE;
END_IF

GetCellData := DataComplete[1] AND DataComplete[2] AND DataComplete[3];
END_METHOD

METHOD GetDiagnostics 
VAR_IN_OUT
	AddError		: ARRAY [*] OF FB_AddErrorST;
	a_ActiveEvents	: ARRAY [*] OF ST_ErrorStruct;
	w_Index			: WORD;
END_VAR
(*BMS errors (sunspec)*)
	(*BMS Communication error*)		AddError[w_Index](
			b_ErrorTrig				:= get.Events.b_COMMUNICATION_ERROR,
			out_ST_Error			:= a_ActiveEvents[w_Index],
			w_ErrorID				:= 1,
			e_ObjectID				:= e_id,						//only first call set object ID.
			s_Message				:= 'communication error',
			e_sev					:= eSeverity.QuickShutdown,	//<-- maybe normal shutdown?
			b_AutoClear				:= FALSE,
			t_TriggerTime			:= TIME#10S,
			e_ErrAckAccess			:= eErrAckAccess.Operator
			);
		w_Index := w_Index +1;
		
	(*Configuration fault*)		AddError[w_Index](
			b_ErrorTrig				:= get.Events.b_CONFIGURATION_ALARM,
			out_ST_Error			:= a_ActiveEvents[w_Index],
			w_ErrorID				:= 2,
			s_Message				:= 'configuration error',
			e_sev					:= eSeverity.NormalShutdown,
			b_AutoClear				:= FALSE,
			e_ErrAckAccess			:= eErrAckAccess.VDL
			//in_t_TriggerTime		:= TIME#500MS,
			//in_e_ErrAckAccess		:= TRUE,
			);
		w_Index := w_Index +1;
	
	(*Configuration warning*)		AddError[w_Index](
			b_ErrorTrig				:= get.Events.b_CONFIGURATION_WARNING,
			out_ST_Error			:= a_ActiveEvents[w_Index],
			w_ErrorID				:= 3,
			s_Message				:= 'configuration error',
			e_sev					:= eSeverity.Warning,
			b_AutoClear				:= FALSE,
			e_ErrAckAccess			:= eErrAckAccess.Operator
			//in_t_TriggerTime		:= TIME#500MS,
			//in_e_ErrAckAccess		:= TRUE,
			);
		w_Index := w_Index +1;
		
	(*Contactor fault*)		AddError[w_Index](
			b_ErrorTrig				:= get.Events.b_CONTACTOR_ERROR,
			out_ST_Error			:= a_ActiveEvents[w_Index],
			w_ErrorID				:= 4,
			s_Message				:= 'contactor fault',
			e_sev					:= eSeverity.QuickShutdown,
			b_AutoClear				:= FALSE,
			e_ErrAckAccess			:= eErrAckAccess.Operator
			//in_t_TriggerTime		:= TIME#500MS,
			//in_e_ErrAckAccess		:= TRUE,
			);
		w_Index := w_Index +1;
		
	(*Current imbalance warning*)		AddError[w_Index](						//unused, will always be false
			b_ErrorTrig				:= get.Events.b_CURRENT_IMBALANCE_WARNING,
			out_ST_Error			:= a_ActiveEvents[w_Index],
			w_ErrorID				:= 5,
			s_Message				:= 'current imbalance warning',
			e_sev					:= eSeverity.Warning,
			b_AutoClear				:= FALSE,
			e_ErrAckAccess			:= eErrAckAccess.General
			//in_t_TriggerTime		:= TIME#500MS,
			);
		w_Index := w_Index +1;
		
	(*Fan error*)		AddError[w_Index](
			b_ErrorTrig				:= get.Events.b_FAN_ERROR,
			out_ST_Error			:= a_ActiveEvents[w_Index],
			w_ErrorID				:= 6,
			s_Message				:= 'fan error',
			e_sev					:= eSeverity.NormalShutdown,
			b_AutoClear				:= FALSE,
			//in_t_TriggerTime		:= TIME#500MS,
			e_ErrAckAccess			:= eErrackAccess.Operator
			);
		w_Index := w_Index +1;

	(*Ground fault*)		AddError[w_Index](
			b_ErrorTrig			:= get.Events.b_GROUND_FAULT,		//unused, will always be false
			out_ST_Error			:= a_ActiveEvents[w_Index],
			w_ErrorID					:= 7,
			s_Message				:= 'insulation fault',
			e_sev					:= eSeverity.Quickshutdown,
			b_AutoClear				:= FALSE,
			//in_t_TriggerTime		:= TIME#500MS,
			//in_e_ErrAckAccess		:= TRUE,
			);
		w_Index := w_Index +1;

	(*Door open error*)		AddError[w_Index](							//unused, will always be false
			b_ErrorTrig			:= get.Events.b_OPEN_DOOR_ERROR,
			out_ST_Error			:= a_ActiveEvents[w_Index],
			w_ErrorID					:= 8,
			s_Message				:= 'door open',
			e_sev					:= eSeverity.NormalShutdown,
			b_AutoClear				:= TRUE,
			//in_t_TriggerTime		:= TIME#500MS,
			//in_e_ErrAckAccess		:= TRUE,
			);
		w_Index := w_Index +1;

	(*misc alarm*)		AddError[w_Index](							
			b_ErrorTrig			:= get.Events.b_OTHER_ALARM,
			out_ST_Error			:= a_ActiveEvents[w_Index],
			w_ErrorID					:= 9,
			s_Message				:= 'miscellaneous error',
			e_sev					:= eSeverity.NormalShutdown,
			b_AutoClear				:= FALSE,
			//in_t_TriggerTime		:= TIME#500MS,
			//in_e_ErrAckAccess		:= TRUE,
			);
		w_Index := w_Index +1;
		
	(*misc warning*)		AddError[w_Index](							
			b_ErrorTrig			:= get.Events.b_OTHER_WARNING,
			out_ST_Error			:= a_ActiveEvents[w_Index],
			w_ErrorID					:= 10,
			s_Message				:= 'miscellaneous warning',
			e_sev					:= eSeverity.Warning,
			b_AutoClear				:= TRUE,
			//in_t_TriggerTime		:= TIME#500MS,
			//in_e_ErrAckAccess		:= TRUE,
			);
		w_Index := w_Index +1;

	(*Overcharge current alarm*)		AddError[w_Index](							
			b_ErrorTrig			:= get.Events.b_OVER_CHARGE_CURRENT_ALARM,
			out_ST_Error			:= a_ActiveEvents[w_Index],
			w_ErrorID					:= 11,
			s_Message				:= 'charge current too high error',
			e_sev					:= eSeverity.NormalShutdown,			
			b_AutoClear				:= FALSE,									
			//in_t_TriggerTime		:= TIME#500MS,
			//in_e_ErrAckAccess		:= TRUE,
			);
		w_Index := w_Index +1;
		
	(*Overcharge current warning*)		AddError[w_Index](							
			b_ErrorTrig			:= get.Events.b_OVER_CHARGE_CURRENT_WARNING,
			out_ST_Error			:= a_ActiveEvents[w_Index],
			w_ErrorID					:= 12,
			s_Message				:= 'charge current high warning',
			e_sev					:= eSeverity.Warning,				//<-- Powerstack should lower the power
			b_AutoClear				:= TRUE,								
			//in_t_TriggerTime		:= TIME#500MS,
			//in_e_ErrAckAccess		:= TRUE,
			);
		w_Index := w_Index +1;
		
	(*OverDischarge current Alarm*)		AddError[w_Index](							
			b_ErrorTrig			:= get.Events.b_OVER_DISCHARGE_CURRENT_ALARM,
			out_ST_Error			:= a_ActiveEvents[w_Index],
			w_ErrorID					:= 13,
			s_Message				:= 'discharge current too high error',
			e_sev					:= eSeverity.NormalShutdown,				
			b_AutoClear				:= FALSE,								
			//in_t_TriggerTime		:= TIME#500MS,
			//in_e_ErrAckAccess		:= TRUE,
			);

		w_Index := w_Index +1;
		
	(*OverDischarge current warning*)		AddError[w_Index](							
			b_ErrorTrig			:= get.Events.b_OVER_DISCHARGE_CURRENT_WARNING,
			out_ST_Error			:= a_ActiveEvents[w_Index],
			w_ErrorID					:= 14,
			s_Message				:= 'discharge current high warning',
			e_sev					:= eSeverity.Warning,				//<-- Powerstack should lower the power
			b_AutoClear				:= TRUE,								
			//in_t_TriggerTime		:= TIME#500MS,
			//in_e_ErrAckAccess		:= TRUE,
			);
		w_Index := w_Index +1;
		
	(*Overcharge r_SOC error*)		AddError[w_Index](							//unused, will remain false
			b_ErrorTrig			:= get.Events.b_OVER_SOC_MAX_ALARM AND NOT st_params.b_DisableSOCAlarm,
			out_ST_Error			:= a_ActiveEvents[w_Index],
			w_ErrorID					:= 15,
			s_Message				:= 'SOC too high error',
			e_sev					:= eSeverity.NormalShutdown,				
			b_AutoClear			:= FALSE,								
			//in_t_TriggerTime		:= TIME#500MS,
			//in_e_ErrAckAccess		:= TRUE,
			);
		w_Index := w_Index +1;
		
	(*Overcharge r_SOC error*)		AddError[w_Index](							//unused, will remain false
			b_ErrorTrig			:= get.Events.b_OVER_SOC_MAX_WARNING,
			out_ST_Error			:= a_ActiveEvents[w_Index],
			w_ErrorID					:= 16,
			s_Message				:= 'SOC high warning',
			e_sev					:= eSeverity.Warning,				
			b_AutoClear				:= TRUE,								
			//in_t_TriggerTime		:= TIME#500MS,
			//in_e_ErrAckAccess		:= TRUE,
			);
		w_Index := w_Index +1;
		
	(*OverDischarge r_SOC error*)		AddError[w_Index](							
			b_ErrorTrig			:= get.Events.b_UNDER_SOC_MIN_ALARM AND NOT st_params.b_DisableSOCAlarm,
			out_ST_Error			:= a_ActiveEvents[w_Index],
			w_ErrorID					:= 17,
			s_Message				:= 'SOC too low error',
			e_sev					:= eSeverity.NormalShutdown,				
			b_AutoClear			:= FALSE,								
			//in_t_TriggerTime		:= TIME#500MS,
			//in_e_ErrAckAccess		:= TRUE,
			);
		w_Index := w_Index +1;
		
	(*OverDischarge r_SOC error*)		AddError[w_Index](							
			b_ErrorTrig			:= get.Events.b_UNDER_SOC_MIN_WARNING,
			out_ST_Error			:= a_ActiveEvents[w_Index],
			w_ErrorID					:= 18,
			s_Message				:= 'SOC low warning',
			e_sev					:= eSeverity.Warning,				
			b_AutoClear				:= TRUE,								
			//in_t_TriggerTime		:= TIME#500MS,
			//in_e_ErrAckAccess		:= TRUE,
			);
		w_Index := w_Index +1;
		
	(*OverTemperature error*)		AddError[w_Index](							
			b_ErrorTrig			:= get.Events.b_OVER_TEMP_ALARM,
			out_ST_Error			:= a_ActiveEvents[w_Index],
			w_ErrorID					:= 19,
			s_Message				:= 'overtemperature alarm',
			e_sev					:= eSeverity.NormalShutdown,				
			b_AutoClear			:= FALSE,
			b_SMSEnableVDL		:= TRUE,								
			//in_t_TriggerTime		:= TIME#500MS,
			//in_e_ErrAckAccess		:= TRUE,
			);
		w_Index := w_Index +1;		

	(*OverTemperature warning*)		AddError[w_Index](							
			b_ErrorTrig			:= get.Events.b_OVER_TEMP_WARNING,
			out_ST_Error			:= a_ActiveEvents[w_Index],
			w_ErrorID					:= 20,
			s_Message				:= 'overtemperature warning',
			e_sev					:= eSeverity.Warning,				
			b_AutoClear			:= FALSE,								
			//in_t_TriggerTime		:= TIME#500MS,
			//in_e_ErrAckAccess		:= TRUE,
			);
		w_Index := w_Index +1;
	
	(*OverVoltage error*)		AddError[w_Index](							
			b_ErrorTrig			:= get.Events.b_OVER_VOLT_ALARM,
			out_ST_Error			:= a_ActiveEvents[w_Index],
			w_ErrorID					:= 21,
			s_Message				:= 'overvoltage error',
			e_sev					:= eSeverity.NormalShutdown,
			b_SMSEnableVDL		:= TRUE,				
			b_AutoClear			:= FALSE,								
			//in_t_TriggerTime		:= TIME#500MS,
			//in_e_ErrAckAccess		:= TRUE,
			);
		w_Index := w_Index +1;		

	(*OverVoltage warning*)		AddError[w_Index](							
			b_ErrorTrig			:= get.Events.b_OVER_VOLT_WARNING,
			out_ST_Error			:= a_ActiveEvents[w_Index],
			w_ErrorID					:= 22,
			s_Message				:= 'overvoltage warning',
			e_sev					:= eSeverity.Warning,				
			b_AutoClear			:= FALSE,								
			//in_t_TriggerTime		:= TIME#500MS,
			//in_e_ErrAckAccess		:= TRUE,
			);
		w_Index := w_Index +1;
		
	(*Temperature imbalance error*)		AddError[w_Index](							
			b_ErrorTrig			:= get.Events.b_TEMPERATURE_IMBALANCE_ALARM,
			out_ST_Error			:= a_ActiveEvents[w_Index],
			w_ErrorID					:= 23,
			s_Message				:= 'temperature imbalance error',
			e_sev					:= eSeverity.NormalShutdown,				
			b_AutoClear			:= FALSE,								
			//in_t_TriggerTime		:= TIME#500MS,
			//in_e_ErrAckAccess		:= TRUE,
			);
		w_Index := w_Index +1;		

	(*Temperature imbalance warning*)		AddError[w_Index](							
			b_ErrorTrig			:= get.Events.b_TEMPERATURE_IMBALANCE_WARNING,
			out_ST_Error			:= a_ActiveEvents[w_Index],
			w_ErrorID					:= 24,
			s_Message				:= 'temperature imbalance warning',
			e_sev					:= eSeverity.Warning,				
			b_AutoClear			:= FALSE,								
			//in_t_TriggerTime		:= TIME#500MS,
			//in_e_ErrAckAccess		:= TRUE,
			);
		w_Index := w_Index +1;

	(*Under Temperature error*)		AddError[w_Index](							
			b_ErrorTrig			:= get.Events.b_UNDER_TEMP_ALARM,
			out_ST_Error			:= a_ActiveEvents[w_Index],
			w_ErrorID					:= 25,
			s_Message				:= 'temperature low error',
			e_sev					:= eSeverity.NormalShutdown,				
			b_AutoClear			:= FALSE,								
			//in_t_TriggerTime		:= TIME#500MS,
			//in_e_ErrAckAccess		:= TRUE,
			);
		w_Index := w_Index +1;		

	(*Under Temperature warning*)		AddError[w_Index](							
			b_ErrorTrig			:= get.Events.b_UNDER_TEMP_WARNING,
			out_ST_Error			:= a_ActiveEvents[w_Index],
			w_ErrorID					:= 26,
			s_Message				:= 'temperature low warning',
			e_sev					:= eSeverity.Warning,				
			b_AutoClear			:= TRUE,								
			//in_t_TriggerTime		:= TIME#500MS,
			//in_e_ErrAckAccess		:= TRUE,
			);
		w_Index := w_Index +1;

	(*Under Temperature error*)		AddError[w_Index](							
			b_ErrorTrig			:= get.Events.b_UNDER_VOLT_ALARM,
			out_ST_Error			:= a_ActiveEvents[w_Index],
			w_ErrorID					:= 27,
			s_Message				:= 'undervoltage error',
			e_sev					:= eSeverity.NormalShutdown,				
			b_AutoClear			:= FALSE,								
			//in_t_TriggerTime		:= TIME#500MS,
			//in_e_ErrAckAccess		:= TRUE,
			);
		w_Index := w_Index +1;		

	(*Under Temperature warning*)		AddError[w_Index](							
			b_ErrorTrig			:= get.Events.b_UNDER_VOLT_WARNING,
			out_ST_Error			:= a_ActiveEvents[w_Index],
			w_ErrorID					:= 28,
			s_Message				:= 'undervoltage warning',
			e_sev					:= eSeverity.Warning,				
			b_AutoClear			:= FALSE,								
			//in_t_TriggerTime		:= TIME#500MS,
			//in_e_ErrAckAccess		:= TRUE,
			);
		w_Index := w_Index +1;
		
	(*Battery voltage imbalance warning*)		AddError[w_Index](							
			b_ErrorTrig			:= get.Events.b_VOLTAGE_IMBALANCE_WARNING,
			out_ST_Error			:= a_ActiveEvents[w_Index],
			w_ErrorID					:= 29,
			s_Message				:= 'voltage imbalance warning',
			e_sev					:= eSeverity.Warning,				
			b_AutoClear			:= FALSE,								
			//in_t_TriggerTime		:= TIME#500MS,
			);
		w_Index := w_Index +1;	
		
		(*Battery voltage imbalance warning*)		AddError[w_Index](							
			b_ErrorTrig			:= get.Events.b_SocHighLimitOutOfRange,
			out_ST_Error			:= a_ActiveEvents[w_Index],
			w_ErrorID					:= 30,
			s_Message				:= 'SOC upper limit out of range',
			e_sev					:= eSeverity.info,				
			b_AutoClear			:= TRUE,								
			);
		w_Index := w_Index +1;	
		
				(*Battery voltage imbalance warning*)		AddError[w_Index](							
			b_ErrorTrig			:= get.Events.b_SocLowLimitOutOfRange,
			out_ST_Error			:= a_ActiveEvents[w_Index],
			w_ErrorID					:= 31,
			s_Message				:= 'SOC lower limit out of range',
			e_sev					:= eSeverity.info,				
			b_AutoClear			:= TRUE,								
			);
		w_Index := w_Index +1;	
	
(*Battery PRECHARGE FAULT*)		AddError[w_Index](							
			b_ErrorTrig			:= get.Events.b_POWERONFAULT,
			out_ST_Error			:= a_ActiveEvents[w_Index],
			w_ErrorID					:= 32,
			s_Message				:= 'precharge fault',
			e_sev					:= eSeverity.warning,				
			b_AutoClear			:= TRUE,								
			);
		w_Index := w_Index +1;	
		
(*Battery power off fault*)		AddError[w_Index](							
			b_ErrorTrig			:= get.Events.b_POWEROFFFAULT,
			out_ST_Error			:= a_ActiveEvents[w_Index],
			w_ErrorID					:= 33,
			s_Message				:= 'poweroff fault',
			e_sev					:= eSeverity.Quickshutdown,				
			b_AutoClear			:= FALSE,								
			);
		w_Index := w_Index +1;	
		
(*Disconnector Off*)		AddError[w_Index](							
			b_ErrorTrig			:= get.Events.b_DISCONNECTOR_OFF,
			out_ST_Error			:= a_ActiveEvents[w_Index],
			w_ErrorID					:= 35,
			s_Message				:= 'HV disconnector(s) off position',
			e_sev					:= eSeverity.Normalshutdown,				
			b_AutoClear			:= FALSE,								
			);
		w_Index := w_Index +1;
		
(*SBMU1 com failed*)		AddError[w_Index](							
			b_ErrorTrig				:= get.Events.b_SBMUCommError[0],
			out_ST_Error			:= a_ActiveEvents[w_Index],
			w_ErrorID				:= 36,
			s_Message				:= 'SBMU 1 Com Warning',
			e_sev					:= eSeverity.Warning,				
			b_AutoClear				:= TRUE,
			t_TriggerTime			:= TIME#5S,								
			);
		w_Index := w_Index +1;

(*SBMU2 com failed*)		AddError[w_Index](							
			b_ErrorTrig				:= get.Events.b_SBMUCommError[1],
			out_ST_Error			:= a_ActiveEvents[w_Index],
			w_ErrorID				:= 37,
			s_Message				:= 'SBMU 2 Com Warning',
			e_sev					:= eSeverity.Warning,				
			b_AutoClear				:= TRUE,
			t_TriggerTime			:= TIME#5S,								
			);
		w_Index := w_Index +1;

(*SBMU3 com failed*)		AddError[w_Index](							
			b_ErrorTrig				:= get.Events.b_SBMUCommError[2],
			out_ST_Error			:= a_ActiveEvents[w_Index],
			w_ErrorID				:= 38,
			s_Message				:= 'SBMU 3 Com Warning',
			e_sev					:= eSeverity.Warning,				
			b_AutoClear				:= TRUE,
			t_TriggerTime			:= TIME#5S,								
			);
		w_Index := w_Index +1;

(*SBMU4 com failed*)		AddError[w_Index](							
			b_ErrorTrig				:= get.Events.b_SBMUCommError[3],
			out_ST_Error			:= a_ActiveEvents[w_Index],
			w_ErrorID				:= 39,
			s_Message				:= 'SBMU 4 Com Warning',
			e_sev					:= eSeverity.Warning,				
			b_AutoClear				:= TRUE,
			t_TriggerTime			:= TIME#5S,								
			);
		w_Index := w_Index +1;
		
(*SBMU1 failed to connect HV*)		AddError[w_Index](							
			b_ErrorTrig				:= get.Events.b_SBMUFailedToConnect[0],
			out_ST_Error			:= a_ActiveEvents[w_Index],
			w_ErrorID				:= 40,
			s_Message				:= 'SBMU 1 failed to connect to DC bus',
			e_sev					:= eSeverity.Warning,				
			b_AutoClear				:= TRUE,
			t_TriggerTime			:= TIME#5S,								
			);
		w_Index := w_Index +1;

(*SBMU2 com failed*)		AddError[w_Index](							
			b_ErrorTrig				:= get.Events.b_SBMUFailedToConnect[1],
			out_ST_Error			:= a_ActiveEvents[w_Index],
			w_ErrorID				:= 41,
			s_Message				:= 'SBMU 2 failed to connect to DC bus',
			e_sev					:= eSeverity.Warning,				
			b_AutoClear				:= TRUE,
			t_TriggerTime			:= TIME#5S,								
			);
		w_Index := w_Index +1;

(*SBMU3 com failed*)		AddError[w_Index](							
			b_ErrorTrig				:= get.Events.b_SBMUFailedToConnect[2],
			out_ST_Error			:= a_ActiveEvents[w_Index],
			w_ErrorID				:= 42,
			s_Message				:= 'SBMU 3 failed to connect to DC bus',
			e_sev					:= eSeverity.Warning,				
			b_AutoClear				:= TRUE,
			t_TriggerTime			:= TIME#5S,								
			);
		w_Index := w_Index +1;

(*SBMU4 com failed*)		AddError[w_Index](							
			b_ErrorTrig				:= get.Events.b_SBMUFailedToConnect[3],
			out_ST_Error			:= a_ActiveEvents[w_Index],
			w_ErrorID				:= 43,
			s_Message				:= 'SBMU 4 failed to connect to DC bus',
			e_sev					:= eSeverity.Warning,				
			b_AutoClear				:= TRUE,
			t_TriggerTime			:= TIME#5S,								
			);
		w_Index := w_Index +1;
		
		
(*SOC too low for conditioning*)		AddError[w_Index](							
			b_ErrorTrig				:= NOT b_InternalHVDCAllowed,
			out_ST_Error			:= a_ActiveEvents[w_Index],
			w_ErrorID				:= 44,
			s_Message				:= 'SOC low warning. Internal Conditioning disabled',
			e_sev					:= eSeverity.Warning,				
			b_AutoClear				:= TRUE,
			t_TriggerTime			:= TIME#5S,								
			);
		w_Index := w_Index +1;
END_METHOD

METHOD PRIVATE GetMBMUData : BOOL
VAR_IN_OUT CONSTANT
	st_params			: ST_BMS_params;
END_VAR


VAR_INST
	
	MBReadMBMU			: 	FB_MBReadRegs;
	MBMUData 			: 	ARRAY[0..52] OF WORD;
	bCommBusy			:	BOOL;
	bComError			:	BOOL;
	errID				:	UDINT;
	cbRead				:	UDINT;
	TransmissionDone	: 	f_trig;
	COMretryCounter		:	USINT := 0;
	//ComTimer			:	Ton := (PT := TIME#100MS);
END_VAR

VAR
	Counter				:	INT;
END_VAR
//read mbmu data every 100ms

GetMBMUData := FALSE;

ComTimer(in := NOT(ComTimer.Q OR bCommBusy));

MBReadMBMU(
sIPAddr := st_params.IP_BMS,
nTCPPort := 502,
nUnitID := 255,//16#FF;
nMBAddr := 0,
nQuantity := 53,
cbLength := SIZEOF(MBMUData),
pDestAddr := ADR(MBMUData),
bExecute := ComTimer.Q,
bBusy => bCommBusy,
bError => bComError,
nErrId => errID,
cbRead => cbRead,
tTimeout := t_TimeOut,
);

TransmissionDone(CLK := bCommBusy);

IF TransmissionDone.Q THEN
	IF NOT bComError THEN
		MEMCPY(ADR(get.MBMU.GeneralSBMUStatus[0]), ADR(MBMUData[0]), 32);	//0x0000 - 0x000f
		MEMCPY(ADR(get.MBMU.MBMUStatus[0]), ADR(MBMUData[16]), 32);			//0x0010 - 0x001f
	
		get.MBMU.BatteryStatus.r_SystemVoltage := WORD_TO_REAL(MBMUData[32])/10; 						//0-1500V with 0.1V/bit
		get.MBMU.BatteryStatus.r_SystemCurrent := WORD_TO_REAL(MBMUData[33])-20000; 					//-20k .. +20k kW in 1kW/bit steps
		
		get.MBMU.BatteryStatus.r_SOC := WORD_TO_REAL(MBMUData[34])/10; 								//0-100% with 0.1%/bit;
		get.MBMU.BatteryStatus.r_SOH := WORD_TO_REAL(MBMUData[35])/10; 								//0-100% with 0.1%/bit;
		
		get.MBMU.BatteryStatus.ar_CellVoltage[eSubValues.Maximum] := WORD_TO_REAL(MBMUData[36])/1000;	//0-5v with 0.001v/bit;
		get.MBMU.BatteryStatus.ar_CellVoltage[eSubValues.Minimum] := WORD_TO_REAL(MBMUData[37])/1000;	//0-5v with 0.001v/bit;
		get.MBMU.BatteryStatus.ar_CellVoltage[eSubValues.Average] := WORD_TO_REAL(MBMUData[38])/1000;	//0-5v with 0.001v/bit;
		
		get.MBMU.BatteryStatus.ar_CellTemperature[eSubValues.Maximum] := WORD_TO_REAL(MBMUData[39])-50;	//-50..200gr with 1gr/bit;
		get.MBMU.BatteryStatus.ar_CellTemperature[eSubValues.Minimum] := WORD_TO_REAL(MBMUData[40])-50;	//-50..200gr with 1gr/bit;
		get.MBMU.BatteryStatus.ar_CellTemperature[eSubValues.Average] := WORD_TO_REAL(MBMUData[41])-50;	//-50..200gr with 1gr/bit;
		
		get.MBMU.BatteryStatus.r_MaxChargeCurrentAllowed := WORD_TO_REAL(MBMUData[42])-20000;			//-20k .. +20k A in 1A/bit steps
		get.MBMU.BatteryStatus.r_MaxDischargeCurrentAllowed := WORD_TO_REAL(MBMUData[43])-20000;			//-20k .. +20k A in 1A/bit steps
		
		get.MBMU.BatteryStatus.r_MaxChargePowerAllowed := WORD_TO_REAL(MBMUData[44])-20000;				//-20k .. +20k kW in 1kW/bit steps
		get.MBMU.BatteryStatus.r_MaxDischargePowerAllowed := WORD_TO_REAL(MBMUData[45])-20000;			//-20k .. +20k kW in 1kW/bit steps
		
		get.MBMU.BatteryStatus.r_SystemPower	:= 	WORD_TO_REAL(MBMUData[46])-20000;						//-20k .. +20k kW in 1kW/bit steps
		get.MBMU.BatteryStatus.r_ChargeSOE	:=	WORD_TO_REAL(MBMUData[47])/10;
		get.MBMU.BatteryStatus.r_DischargeSOE	:=	WORD_TO_REAL(MBMUData[48])/10;
		
		get.MBMU.BatteryStatus.r_RemainingChargeEnergy	:=	WORD_TO_REAL(MBMUData[49]) *2;
		get.MBMU.BatteryStatus.r_RemainingDischargeEnergy	:=	WORD_TO_REAL(MBMUData[50]) *2;
		
		get.MBMU.BatteryStatus.r_MaxSystemVoltageAllowed := WORD_TO_REAL(MBMUData[51])/10; 			//0-1500V with 0.1V/bit
		get.MBMU.BatteryStatus.r_MinSystemVoltageAllowed := WORD_TO_REAL(MBMUData[52])/10; 			//0-1500V with 0.1V/bit
			
		memcpy(ADR(arDatalogMBMU), ADR(MBMUData), 92);	//0-46
		
		GetMBMUData := TRUE;
		COMretryCounter := 0;
		b_MBComErrorActive := FALSE;
	ELSE
		COMretryCounter := COMretryCounter +1;
		IF COMRetryCounter > 5 THEN
			b_MBComErrorActive := TRUE;
		END_IF
	END_IF
END_IF
END_METHOD

METHOD PRIVATE GetMBMUStaticSystemData : BOOL
VAR_IN_OUT CONSTANT
	st_params			: ST_BMS_params;
END_VAR

VAR_INST
	MBReadBMS			: 	FB_MBReadRegs;
	DataBuffer 			: 	ARRAY[0..31] OF WORD;
	
	bCommBusy			:	BOOL;
	bComError			:	BOOL;
	errID				:	UDINT;
	cbRead				:	UDINT;
	
	TransmissionDone 	: 	f_trig;
	COMretryCounter		:	USINT := 0;
	//ComTimer			:	Ton := (PT := TIME#200ms);
END_VAR

//Read ETH+MBMU SW/HW version at init.
GetMBMUStaticSystemData := FALSE;

ComTimer(in := NOT(ComTimer.Q));

MBReadBMS(
sIPAddr := st_params.IP_BMS,
nTCPPort := 502,
nUnitID := 255,//16#FF;
nMBAddr := 256,
nQuantity := 32,
cbLength := SIZEOF(DataBuffer),
pDestAddr := ADR(DataBuffer),
bExecute := ComTimer.Q,
tTimeout := t_TimeOut,
bBusy => bCommBusy,
bError => bComError,
nErrId => errID,
cbRead => cbRead
);

TransmissionDone(CLK := bCommBusy);

IF TransmissionDone.Q THEN
	IF NOT bComError THEN
		memcpy(destAddr := ADR(get.MBMU.s_MBMU_SWVer), SrcAddr := ADR(DataBuffer[0]), n := 16);
		memcpy(destAddr  := ADR(get.MBMU.s_MBMU_HWVer), SrcAddr := ADR(DataBuffer[8]), n := 16);
		memcpy(destAddr  := ADR(get.MBMU.s_ETH_SWVer), SrcAddr := ADR(DataBuffer[16]), n := 16);
		memcpy(destAddr  := ADR(get.MBMU.r_ETH_HWVer), SrcAddr :=ADR( DataBuffer[24]), n := 16);
		GetMBMUStaticSystemData := TRUE;
		COMretryCounter := 0;
		b_MBComErrorActive := FALSE;
	ELSE
		COMretryCounter := COMretryCounter +1;
		IF COMRetryCounter > 5 THEN
			b_MBComErrorActive := TRUE;
		END_IF
	END_IF
END_IF
END_METHOD

METHOD PRIVATE GetSBMUData : BOOL
VAR_IN_OUT CONSTANT
	st_params			: ST_BMS_params;
END_VAR

VAR_INST
	MBReadSBMU		: 	FB_MBReadRegs;
	DataBuffer		:	ARRAY[0..91] OF WORD;
	bCommBusy		:	BOOL;
	bComError		:	BOOL;
	errID			:	UDINT;
	cbRead			:	UDINT;
	CommDone		: 	f_trig;
	tempSBMUStatus	:	WORD;
	SBMUCounter		: 	USINT	:=	0;
	//ComTimer			:	Ton := (PT := TIME#100MS);
END_VAR

VAR
	b_MainRelayClosed 		: 	BOOL;
	b_PrechargeRelayClosed	:	BOOL;
	ui_SBMUCounter			:	uint;
END_VAR
GetSBMUData := FALSE;

ComTimer(in := NOT(ComTimer.Q OR bCommbusy));

MBReadSBMU(
	sIPAddr := st_params.IP_BMS,
	nTCPPort := 502,
	nUnitID := 255,//16#FF;
	nMBAddr := 1024*(SBMUcounter+1),
	nQuantity := 91,
	cbLength := SIZEOF(DataBuffer),
	pDestAddr := ADR(DataBuffer),
	bExecute := ComTimer.Q,
	tTimeout := t_TimeOut,
	bBusy => bCommBusy,
	bError => bComError,
	nErrId => errID,
	cbRead => cbRead
);
	
CommDone(CLK := bCommBusy);
	
IF CommDone.Q THEN
	IF NOT bComError THEN
		get.SBMU[SBMUcounter].w_SystemWarning := DataBuffer[0];
		get.SBMU[SBMUcounter].SystemAlarm[0] := DataBuffer[1];
		get.SBMU[SBMUcounter].SystemAlarm[1] := DataBuffer[2];
		get.SBMU[SBMUcounter].SystemAlarm[2] := DataBuffer[3];
		
		get.SBMU[SBMUcounter].b_PrechargeRelayClosed 	:= WORD_TO_BOOL(DataBuffer[16]);
		get.SBMU[SBMUcounter].b_MainPosRelayClosed	 	:= WORD_TO_BOOL(DataBuffer[17]);
		get.SBMU[SBMUcounter].b_MainNegRelayClosed		:= WORD_TO_BOOL(DataBuffer[18]);
		get.SBMU[SBMUcounter].b_ControlBoxFanOn 			:= WORD_TO_BOOL(DataBuffer[19]);
		get.SBMU[SBMUcounter].b_BalanceStatus 			:= WORD_TO_BOOL(DataBuffer[20]);
		
		get.SBMU[SBMUcounter].BatteryStatus.r_SystemVoltage := WORD_TO_REAL(DataBuffer[32])/10;	//0-1500V with 0.1V/bit
		get.SBMU[SBMUcounter].BatteryStatus.r_SystemCurrent := (WORD_TO_REAL(DataBuffer[34])/10)-2000; 	//-2k .. +2k A in 0.1A/bit steps
		
		get.SBMU[SBMUcounter].BatteryStatus.r_SOC := WORD_TO_REAL(DataBuffer[35])/10; 			//0-100% with 0.1%/bit;
		get.SBMU[SBMUcounter].BatteryStatus.r_SOH := WORD_TO_REAL(DataBuffer[36])/10;				//0-100% with 0.1%/bit;
		
		get.SBMU[SBMUcounter].BatteryStatus.ar_CellVoltage[eSubValues.Maximum] := WORD_TO_REAL(DataBuffer[37])/1000;	//0-5v with 0.001v/bit;
		get.SBMU[SBMUcounter].BatteryStatus.ar_CellVoltage[eSubValues.Minimum] := WORD_TO_REAL(DataBuffer[38])/1000;	//0-5v with 0.001v/bit;
		get.SBMU[SBMUcounter].BatteryStatus.ar_CellVoltage[eSubValues.Average] := WORD_TO_REAL(DataBuffer[39])/1000;	//0-5v with 0.001v/bit;
		
		get.SBMU[SBMUcounter].BatteryStatus.ar_CellTemperature[eSubValues.Maximum] := WORD_TO_REAL(DataBuffer[40])-50;	//-50..200gr with 1gr/bit;
		get.SBMU[SBMUcounter].BatteryStatus.ar_CellTemperature[eSubValues.Minimum] := WORD_TO_REAL(DataBuffer[41])-50;	//-50..200gr with 1gr/bit;
		get.SBMU[SBMUcounter].BatteryStatus.ar_CellTemperature[eSubValues.Average] := WORD_TO_REAL(DataBuffer[42])-50;	//-50..200gr with 1gr/bit;
		
		get.SBMU[SBMUcounter].BatteryStatus.r_MaxChargeCurrentAllowed := 		(WORD_TO_REAL(DataBuffer[43])/10)-2000;	//-2k .. +2k A in 0.1A/bit steps
		get.SBMU[SBMUcounter].BatteryStatus.r_MaxDischargeCurrentAllowed := 		(WORD_TO_REAL(DataBuffer[44])/10)-2000;	//-2k .. +2k A in 0.1A/bit steps
		
		get.SBMU[SBMUcounter].BatteryStatus.w_MaxVoltageCellLocation := DataBuffer[48];
		get.SBMU[SBMUcounter].BatteryStatus.w_MinVoltageCellLocation := DataBuffer[49];
		
		get.SBMU[SBMUcounter].BatteryStatus.w_MaxTempCellLocation := DataBuffer[50];
		get.SBMU[SBMUcounter].BatteryStatus.w_MinTempCellLocation := DataBuffer[51];
	
		
		//Collect dataset for CATL datalog
		memcpy(ADR(arDatalogSBMU[SBMUcounter][0]), ADR(DataBuffer[0]), 32); 	//0-15
		tempSBMUStatus.0		:= WORD_TO_BOOL(DataBuffer[16]);
		tempSBMUStatus.1	 	:= WORD_TO_BOOL(DataBuffer[17]);
		tempSBMUStatus.2		:= WORD_TO_BOOL(DataBuffer[18]);
		tempSBMUStatus.3 		:= WORD_TO_BOOL(DataBuffer[19]);
		tempSBMUStatus.4 		:= WORD_TO_BOOL(DataBuffer[20]); 
		tempSBMUStatus.5 		:= WORD_TO_BOOL(DataBuffer[21]);
		arDatalogSBMU[SBMUcounter][16] := tempSBMUStatus;						//16
		memcpy(ADR(arDatalogSBMU[SBMUcounter][17]), ADR(DataBuffer[32]), 44);	//17-38
		arDatalogSBMU[SBMUcounter][39] := DataBuffer[56];						//39
		arDatalogSBMU[SBMUcounter][40] := DataBuffer[57];						//40
		arDatalogSBMU[SBMUcounter][41] := DataBuffer[58];						//41
		arDatalogSBMU[SBMUcounter][42] := DataBuffer[59];						//42
		memcpy(ADR(arDatalogSBMU[SBMUcounter][43]), ADR(DataBuffer[54]), 16);	//43

	(* GIVES RUNTIME EXCEPTION !!! NaN value coming from bms making a runtime exception*)
		//MEMCPY(ADR(get.SBMU[SBMUcounter].BatteryStatus.r_HistAccChargeEnergy), ADR(DataBuffer[85]), 2);  // low word
		//MEMCPY(ADR(get.SBMU[SBMUcounter].BatteryStatus.r_HistAccChargeEnergy)+2, ADR(DataBuffer[84]), 2);  // high word
		//get.SBMU[SBMUcounter].BatteryStatus.r_HistAccChargeEnergy := get.SBMU[SBMUcounter].BatteryStatus.r_HistAccChargeEnergy/10; //0-449GHW with 0.1kWh/bit
		
		//MEMCPY(ADR(get.SBMU[SBMUcounter].BatteryStatus.r_HistAccDischargeEnergy), ADR(DataBuffer[87]), 2);  // low word
		//MEMCPY(ADR(get.SBMU[SBMUcounter].BatteryStatus.r_HistAccDischargeEnergy)+2, ADR(DataBuffer[86]), 2);  // high word
		//get.SBMU[SBMUcounter].BatteryStatus.r_HistAccDischargeEnergy := get.SBMU[SBMUcounter].BatteryStatus.r_HistAccDischargeEnergy/10; //0-449GHW with 0.1kWh/bit
	
		
		get.events.b_SBMUCommError[SBMUCounter] := FALSE;
		
		SBMUCounter := SBMUCounter +1;
		
		IF SBMUCounter >= by_NoOfStrings THEN//BMSGet.MBMU_Status.by_NumberOfSubSystems THEN
			GetSBMUData := TRUE;
			SBMUCounter := 0;
		END_IF
		
		IF 		(get.SBMU[0].b_MainPosRelayClosed AND get.SBMU[0].b_MainNegRelayClosed) OR 
				(get.SBMU[1].b_MainPosRelayClosed AND get.SBMU[1].b_MainNegRelayClosed) OR
				(get.SBMU[2].b_MainPosRelayClosed AND get.SBMU[2].b_MainNegRelayClosed) OR
				(get.SBMU[3].b_MainPosRelayClosed AND get.SBMU[3].b_MainNegRelayClosed) THEN
			PowerStatus := eHVDC_PowerStatus.On;
		ELSIF 	get.SBMU[0].b_PrechargeRelayClosed OR 
				(get.SBMU[1].b_PrechargeRelayClosed AND (by_NoOfStrings > 1)) OR 
				(get.SBMU[2].b_PrechargeRelayClosed AND (by_NoOfStrings > 2))  OR 
				(get.SBMU[3].b_PrechargeRelayClosed AND (by_NoOfStrings > 3)) THEN
			PowerStatus := eHVDC_PowerStatus.Precharging;
		ELSE
			PowerStatus := eHVDC_PowerStatus.Off;
		END_IF	
		
		get.events.b_SBMUFailedToConnect[0] := PowerStatus = eHVDC_PowerStatus.On AND NOT (get.SBMU[0].b_MainPosRelayClosed AND get.SBMU[0].b_MainNegRelayClosed);
		get.events.b_SBMUFailedToConnect[1] := PowerStatus = eHVDC_PowerStatus.On AND (NOT (get.SBMU[1].b_MainPosRelayClosed AND get.SBMU[1].b_MainNegRelayClosed)) AND by_NoOfStrings > 1;
		get.events.b_SBMUFailedToConnect[2] := PowerStatus = eHVDC_PowerStatus.On AND (NOT (get.SBMU[2].b_MainPosRelayClosed AND get.SBMU[2].b_MainNegRelayClosed)) AND by_NoOfStrings > 2;
		get.events.b_SBMUFailedToConnect[3] := PowerStatus = eHVDC_PowerStatus.On AND (NOT (get.SBMU[3].b_MainPosRelayClosed AND get.SBMU[3].b_MainNegRelayClosed)) AND by_NoOfStrings > 3;
		
	ELSE
		get.events.b_SBMUCommError[SBMUCounter] := TRUE;
		SBMUCounter := SBMUCounter +1;
	END_IF
END_IF
END_METHOD

METHOD PRIVATE GetSBMUStaticSystemData : BOOL
VAR_IN_OUT CONSTANT
	st_params			: ST_BMS_params;
END_VAR


VAR_INPUT
	SBMU_ID				:	uint;	
END_VAR

VAR_INST
	MBReadBMS			: 	FB_MBReadRegs;
	DataBuffer 			: 	ARRAY[0..31] OF WORD;
	
	bCommBusy			:	BOOL;
	bComError			:	BOOL;
	errID				:	UDINT;
	cbRead				:	UDINT;
	
	TransmissionDone 	: 	f_trig;
	ComretryCounter		:	USINT := 0;
	
	//ComTimer			:	Ton := (PT := TIME#0S200MS);
END_VAR


VAR
	SBMU: INT;
END_VAR
//Read ETH+MBMU SW/HW version at init.
GetSBMUStaticSystemData := FALSE;

IF (SBMU_ID<1) OR (SBMU>4)then //BMSGET.MBMU_Status.by_NumberOfSubSystems) THEN
	GetSBMUStaticSystemData := TRUE;
	RETURN;
END_IF

ComTimer(in := NOT(ComTimer.Q OR bCommbusy));

MBReadBMS(
sIPAddr := st_params.IP_BMS,
nTCPPort := 502,
nUnitID := 255,//16#FF;
nMBAddr := 960 + (SBMU_ID*1024),
nQuantity := 32,
cbLength := SIZEOF(DataBuffer),
pDestAddr := ADR(DataBuffer),
bExecute := ComTimer.Q,
tTimeout := t_TimeOut,
bBusy => bCommBusy,
bError => bComError,
nErrId => errID,
cbRead => cbRead
);

TransmissionDone(CLK := bCommBusy);

IF TransmissionDone.Q THEN
	IF NOT bComError THEN
	//werkt niet. Bij de MBMU gek genoeg wel
	//	memcpy(destAddr := ADR(BMSGet.SBMU[SBMU_ID].s_SBMU_SWVer), SrcAddr := ADR(DataBuffer[0]), n := 16);
	//	memcpy(destAddr  := ADR(BMSGet.SBMU[SBMU_ID].s_SBMU_HWVer), SrcAddr := ADR(DataBuffer[8]), n := 16);
	//	memcpy(destAddr  := ADR(BMSGet.SBMU[SBMU_ID].s_CSC_SWVer), SrcAddr := ADR(DataBuffer[16]), n := 16);
	//	memcpy(destAddr  := ADR(BMSGet.SBMU[SBMU_ID].s_CSC_HWVer), SrcAddr := ADR(DataBuffer[24]), n := 16);
		GetSBMUStaticSystemData := TRUE;
		get.events.b_SBMUCommError[SBMU_ID] := FALSE;
	ELSE
		get.events.b_SBMUCommError[SBMU_ID] := TRUE;
	END_IF
END_IF
END_METHOD

METHOD PRIVATE GetSystemStatus : BOOL
VAR_IN_OUT CONSTANT
	st_params			: ST_BMS_params;
END_VAR

VAR_INST
	MBReadBMS			: 	FB_MBReadRegs;
	DataBuffer 			: 	ARRAY[0..5] OF WORD;
	
	bCommBusy			:	BOOL;
	bComError			:	BOOL;
	errID				:	UDINT;
	cbRead				:	UDINT;
	
	TransmissionDone 	: 	f_trig;
	
	//ComTimer			:	Ton := (PT := TIME#0S200MS);
	
	ComretryCounter	:	USINT := 0;
END_VAR

//Read general BMS status
GetSystemStatus := FALSE;

ComTimer(in := NOT (ComTimer.Q OR bCommBusy));

MBReadBMS(
sIPAddr := st_params.IP_BMS,
nTCPPort := 502,
nUnitID := 255,//16#FF;
nMBAddr := 769,
nQuantity := 6,
cbLength := SIZEOF(DataBuffer),
pDestAddr := ADR(DataBuffer),
bExecute := ComTimer.Q,
bBusy => bCommBusy,
bError => bComError,
nErrId => errID,
cbRead => cbRead,
tTimeout := t_TimeOut,
);

TransmissionDone(CLK := bCommBusy);

IF TransmissionDone.Q THEN
	IF NOT bComError THEN
		CASE DataBuffer[0] OF
			0: get.MBMU.BatteryStatus.e_BMS_PowerOnStatus := ePowerOnStatus.Off;
			1: get.MBMU.BatteryStatus.e_BMS_PowerOnStatus := ePowerOnStatus.On;
			2: get.MBMU.BatteryStatus.e_BMS_PowerOnStatus := ePowerOnStatus.PowerOn_Fault;
			3: get.MBMU.BatteryStatus.e_BMS_PowerOnStatus := ePowerOnStatus.PowerOff_Fault;
		END_CASE
		
		get.BatteryInfo.e_BMS_PowerOnStatus := get.MBMU.BatteryStatus.e_BMS_PowerOnStatus;
		
		CASE DataBuffer[1] OF
			0: get.MBMU.BatteryStatus.e_BMS_Status := eBMS_Status.Init;
			1: get.MBMU.BatteryStatus.e_BMS_Status := eBMS_Status.Normal;
			2: get.MBMU.BatteryStatus.e_BMS_Status := eBMS_Status.FullCharge;
			3: get.MBMU.BatteryStatus.e_BMS_Status := eBMS_Status.FullDischarge;
			4: get.MBMU.BatteryStatus.e_BMS_Status := eBMS_Status.Warning;
			5: get.MBMU.BatteryStatus.e_BMS_Status := eBMS_Status.Fault;
		END_CASE
		
		get.BatteryInfo.e_BMS_Status := get.MBMU.BatteryStatus.e_BMS_Status;
		
		arDatalogMBMU[48] := DataBuffer[0];
		arDatalogMBMU[49] := DataBuffer[1];
		arDatalogMBMU[50] := DataBuffer[3];
		arDatalogMBMU[51] := DataBuffer[4];
		arDatalogMBMU[52] := DataBuffer[5];	

		
		get.MBMU.by_NumberOfSubSystems := WORD_TO_BYTE(DataBuffer[3]);
		GetSystemStatus := TRUE;
		ComretryCounter := 0;
		b_MBComErrorActive := FALSE;
	ELSE
		COMretryCounter := COMretryCounter +1;
		IF COMRetryCounter > 5 THEN
			b_MBComErrorActive := TRUE;
		END_IF
	END_IF
END_IF
END_METHOD

METHOD GetWearCounters : BOOL
VAR_INST
	PowerOnTimeLogger		:	FB_Varlogger;
	PowerOnCycleLogger		:	FB_Varlogger;
	PrechargeCycleLogger	:	FB_Varlogger;
	OvertempCountLogger		:	FB_Varlogger;
	OverTempTimeLogger		:	FB_Varlogger;
	UnderTempCountLogger	:	FB_Varlogger;
	UnderTempTimeLogger		:	FB_Varlogger;
	
	SlowDataTimer				:	TON := (PT := T#2M);
	rtrig_SOCCalibrationDone	: 	r_trig;
	ton_prechargeDelay			:	ton := (Pt := T#30S);
	
	LastCalibrationTime		:	STRING;
END_VAR
//only log data when BMS communication is actually working
SlowDataTimer(in := NOT SlowDataTimer.q AND BMSDataValid);

PowerOnTimeLogger(		TriggerInput := get.BatteryInfo.e_BMS_PowerOnStatus = ePowerOnStatus.On, 
						LogItemGroup :=  eLogItemGroupID.BMS, 
						LogItemName := 'HVOnHrs', 
						LogType := eLogTypes.TrackOnTime);

PowerOnCycleLogger(		TriggerInput := PowerStatus = eHVDC_PowerStatus.ON, 
						LogItemGroup :=  eLogItemGroupID.BMS, 
						LogItemName := 'HvOnCnt', 
						LogType := eLogTypes.TrackCycles);	

PrechargeCycleLogger(	TriggerInput := PowerStatus = eHVDC_PowerStatus.Precharging, 
						LogItemGroup :=  eLogItemGroupID.BMS, 
						LogItemName := 'PrechargeCnt', 
						LogType := eLogTypes.TrackCycles);	
												
OvertempCountLogger(	TriggerInput := get.Events.b_OVER_TEMP_WARNING, 
						LogItemGroup :=  eLogItemGroupID.BMS, 
						LogItemName := 'OverTempCnt', 
						LogType := eLogTypes.TrackCycles);	

OverTempTimeLogger(		TriggerInput := get.Events.b_OVER_TEMP_WARNING, 
						LogItemGroup :=  eLogItemGroupID.BMS, 
						LogItemName := 'OverTempHrs', 
						LogType := eLogTypes.TrackOnTime);			

UndertempCountLogger(	TriggerInput := get.Events.b_UNDER_TEMP_WARNING, 
						LogItemGroup :=  eLogItemGroupID.BMS, 
						LogItemName := 'UnderTempCnt', 
						LogType := eLogTypes.TrackCycles);	

UnderTempTimeLogger(	TriggerInput := get.Events.b_UNDER_TEMP_WARNING, 
						LogItemGroup :=  eLogItemGroupID.BMS, 
						LogItemName := 'UnderTempHrs', 
						LogType := eLogTypes.TrackOnTime);	

IF BMSDataValid THEN 
	Wearlogging.SetFloat(	eLogItemGroupID.BMS, 	'BattSOH', 				eLogTypes.WriteValue, 			REAL_TO_LREAL(get.BatteryInfo.r_SOH));
	Wearlogging.SetInteger(	eLogItemGroupID.BMS, 	'BattCycles', 			eLogTypes.WriteValue, 			UINT_TO_LINT(get.BatteryInfo.ui_CycleCount));
	Wearlogging.SetFloat(	eLogItemGroupID.BMS, 	'EnergyIn', 			eLogTypes.KeepHighestValue, 	REAL_TO_LREAL(get.BatteryInfo.r_HistAccChargeEnergy));
	Wearlogging.SetFloat(	eLogItemGroupID.BMS, 	'EnergyOut', 			eLogTypes.KeepHighestValue, 	REAL_TO_LREAL(get.BatteryInfo.r_HistAccDischargeEnergy));
	Wearlogging.SetFloat(	eLogItemGroupID.BMS, 	'MaxTempEver', 			eLogTypes.KeepHighestValue, 	REAL_TO_LREAL(get.BatteryInfo.ar_CellTemperature[eSubValues.Maximum]));
	
	IF get.BatteryInfo.ar_CellTemperature[eSubValues.Minimum] > -50 THEN
		Wearlogging.SetFloat(	eLogItemGroupID.BMS, 	'MinTempEver', 			eLogTypes.KeepLowestValue, 		REAL_TO_LREAL(get.BatteryInfo.ar_CellTemperature[eSubValues.Minimum]));
	END_IF
	
	Wearlogging.SetFloat(	eLogItemGroupID.BMS, 	'MaxStringVoltageEver', eLogTypes.KeepHighestValue, 	REAL_TO_LREAL(get.BatteryInfo.r_maxVoltageEver));
END_IF

ton_prechargeDelay(in := get.BatteryInfo.e_BMS_PowerOnStatus = ePowerOnStatus.On);
IF ton_prechargeDelay.Q THEN
	Wearlogging.SetFloat(	eLogItemGroupID.BMS, 	'MinStringVoltageEver', 		eLogTypes.KeepLowestValue, 	REAL_TO_LREAL(get.BatteryInfo.r_SystemVoltage));
END_IF


rtrig_SOCCalibrationDone(clk := get.BatteryInfo.e_BMS_Status = eBMS_Status.FullCharge);		
IF rtrig_SOCCalibrationDone.Q THEN
	dt_LastCalibrationDate := gvl.dt_SystemDateTime;
	LastCalibrationTime:= DT_TO_STRING(gvl.dt_SystemDateTime);
	Wearlogging.SetString(eLogItemGroupID.BMS, 'LastSocCalibration', 	LastCalibrationTime);
END_IF

IF slowDataTimer.Q THEN
	slowDataTimer.Q;
END_IF
							
//Add: Last calibration date
END_METHOD

METHOD Init : BOOL
VAR_INPUT
END_VAR

VAR
	temp1	:	LREAL;
	temp2	:	LREAL;
END_VAR
IF NOT InitDone THEN
	Wearlogging.GetFloatValue(eLogItemGroupID.BMS, 	'EnergyIn', CurrentLogValue => temp1);
	get.BatteryInfo.r_HistAccDischargeEnergy := LREAL_TO_REAL(temp1);
	get.MBMU.BatteryStatus.r_HistAccDischargeEnergy := LREAL_TO_REAL(temp1);
	
	Wearlogging.GetFloatValue(eLogItemGroupID.BMS, 	'EnergyOut', CurrentLogValue => temp2);
	
	get.BatteryInfo.r_HistAccChargeEnergy := LREAL_TO_REAL(temp2);
	get.MBMU.BatteryStatus.r_HistAccChargeEnergy := LREAL_TO_REAL(temp2);

	Wearlogging.SetInteger(	eLogItemGroupID.BMS, 	'nameplateEnergyCapacity', 			eLogTypes.WriteValue, 			REAL_TO_LINT(Settings.Properties.r_RatedEnergyCapacity));
	InitDone := TRUE;
END_IF
END_METHOD

METHOD PRIVATE OpenInsulationSwitch : BOOL
VAR_IN_OUT CONSTANT
	st_params			: ST_BMS_params;
END_VAR

VAR_INPUT
	OpenSwitch : BOOL;
END_VAR

VAR_INST
	WriteReg	:	FB_MBWriteSingleReg;
	Value 		:	WORD 	:= 0;
	StartWrite	:	BOOL	:= FALSE;
	
	bCommBusy	:	BOOL;
	bComError	:	BOOL;
	errID		:	UDINT;

	TransmissionDone 	: 	f_trig;
	ComRetryCounter	:	USINT;
	
	ComTimer			:	Ton := (PT := TIME#0S200MS);
END_VAR

ComTimer(in := NOT(ComTimer.Q));

OpenInsulationswitch := FALSE;

IF OpenSwitch THEN
	Value := 1;
ELSE
	Value := 0;
END_IF

WriteReg(
sIPAddr := st_params.IP_BMS,
nTCPPort := 502,
nUnitID := 255,//16#FF;
nMBAddr := 907,
nValue := Value,
tTimeout := T#0S100MS,
bExecute := ComTimer.q,
bBusy => bCommBusy,
bError => bComError,
nErrId => errID,
);

TransmissionDone(CLK := bCommBusy);

IF TransmissionDone.Q THEN
	IF NOT bComError THEN
		arDatalogEMS[3] := 1;	
		get.MBMU.b_InsulationSwitchOpen := OpenSwitch;
		ComRetryCounter := 0;
		OpenInsulationSwitch := TRUE;
		b_MBComErrorActive := FALSE;
	ELSE
		COMretryCounter := COMretryCounter +1;
		IF COMRetryCounter > 5 THEN
			b_MBComErrorActive := TRUE;
		END_IF
	END_IF
END_IF
END_METHOD

METHOD Reset : BOOL
VAR_INPUT
	//BMSSET	:	st_BMS_Set;
	//ResetIn	:	BOOL;
END_VAR

VAR_INST
	ResetTrigger		:	Ton := (PT := TIME#1S0MS);
	ResetVar			:	BOOL;
END_VAR
b_MBComErrorActive := FALSE;
Reset := ClearBMSFaults(st_params);

FBState := ePOUState.Normal;
END_METHOD

METHOD PRIVATE SetBMSDateTime : BOOL
VAR_IN_OUT CONSTANT
	st_params			: ST_BMS_params;
END_VAR

VAR
	SystemTimeData	:	Timestruct;
	RTCData	:	ARRAY[0..6] OF WORD;	
	
END_VAR
VAR_INST
	//ComTimer			:	Ton := (PT := TIME#0S200MS);
	WriteRegs		:	FB_MBWriteRegs;
	SystemTime		:	FB_LocalSystemTime;
	TransmissionDone 	: 	f_trig;
	SystemTimeDataValid	:	BOOL;
	bCommBusy		:	BOOL;
	bComError		:	BOOL;
	errID			:	UDINT;
	COMRetryCounter	:	USINT := 0;
END_VAR
ComTimer(in := NOT(ComTimer.Q OR bCommBusy));

//write PLC system time to BMS RTC
SetBMSDateTime := FALSE;


//retrieve system time struct
SystemTime(
	sNetID := '',
	bEnable := TRUE,
	dwCycle := 1,
	dwOpt	:= 1,
	tTimeout := t_TimeOut,
	bValid => SystemtimeDataValid,
	systemTime => SystemTimeData
);

//parse system time to BMS data array
IF SystemTimeDataValid THEN
	RTCData[0] := 2024;//SystemTimeData.wYear;
	RTCData[1] := 03;//SystemTimeData.wMonth;
	RTCData[2] := 26;//SystemTimeData.wDay;
	RTCData[3] := 13;//SystemTimeData.wHour;
	RTCData[4] := 52;//SystemTimeData.wMinute;
	RTCData[5] := 00;//SystemTimeData.wSecond;
	RTCData[6] := 1;//can this value remain at 1? or reset to 0 after write?
	
	//write data to BMS
	WriteRegs(	
	sIPAddr := st_params.IP_BMS,
	nTCPPort := 502,
	nUnitID := 255,//16#FF;
	nMBAddr := 900,
	nQuantity := 7,
	pSrcAddr := ADR(RTCData),
	cbLength := SIZEOF(RTCData),
	bExecute := ComTimer.Q,
	tTimeout := TIME#100MS,
	bBusy => bCommBusy,
	bError => bComError,
	nErrId => errID,
	);
	
	TransmissionDone(CLK := bCommBusy);
	
	//return true if tranmission succeeds
	IF TransmissionDone.Q THEN
		IF NOT bComError THEN
			SetBMSDateTime := TRUE;
			ComRetryCounter := 0;
			b_MBComErrorActive := FALSE;
		ELSE
			COMretryCounter := COMretryCounter +1;
			IF COMRetryCounter > 5 THEN
				b_MBComErrorActive := TRUE;
			END_IF
		END_IF
	END_IF
END_IF
END_METHOD

METHOD PRIVATE SetPowerMode : BOOL
VAR_IN_OUT CONSTANT
	st_params			: ST_BMS_params;
END_VAR

VAR_INST
	WriteReg	:	FB_MBWriteSingleReg;
	Value 		:	WORD 	:= 1;
	StartWrite	:	BOOL	:= FALSE;
	bCommBusy	:	BOOL;
	bComError	:	BOOL;
	errID		:	UDINT;
	TransmissionDone 	: 	f_trig;
	//ComTrigger	:	Ton := (PT := TIME#200MS);
	ComRetryCounter	:	USINT	:= 0;
	
	b_HVRequest			: BOOL;
	ton_StartRetrigger	: ton :=(PT := T#5S);
END_VAR	

VAR_INST
	rtrigPowerOn		: R_trig;
END_VAR

//Value := ePowerControl.Stay; //default command is: Do nothing
//it may also work if we just keep sending "poweron" if b_HVDC_Required is true. But this doesn't seem to be the way they intended.
b_HVRequest := b_HVDC_OnRq AND NOT ton_StartRetrigger.Q AND get.BatteryInfo.e_BMS_PowerOnStatus <> ePowerOnSTatus.On;
ton_StartRetrigger(IN:=b_HVRequest);
rtrigPowerOn(CLK:= ton_StartRetrigger.Q);



IF NOT b_HVDC_OnRq AND get.BatteryInfo.e_BMS_PowerOnStatus <> ePowerOnSTatus.Off THEN
	Value := ePowerControl.PowerOff;
ELSIF rtrigPowerOn.Q THEN
	Value := ePowerControl.PowerOn;
END_IF

//Write this register every second, regardless of change.
ComTimer(in := NOT(ComTimer.Q OR bCommBusy));

//IF BMSGet.BattInfo.ui_BMS_Status < 5 THEN
WriteReg(
	sIPAddr := st_params.IP_BMS,
	nTCPPort := 502,
	nUnitID := 255,//16#FF;
	nMBAddr := 897,
	nValue := Value,
	tTimeout := t_TimeOut,
	bExecute := ComTimer.Q,
	bBusy => bCommBusy,
	bError => bComError,
	nErrId => errID,
);
//ELSE
//	SetPowerMode := TRUE;
//END_IF

TransmissionDone(CLK := bCommBusy);
	
//return true if tranmission succeeds
IF TransmissionDone.Q THEN
	IF NOT bComError THEN
		arDatalogEMS[1] := Value;	
	
		SetPowerMode := TRUE;
		ComRetryCounter := 0;
		Value := ePowerControl.Stay;
		b_MBComErrorActive := FALSE;
	ELSE
		COMretryCounter := COMretryCounter +1;
		IF COMRetryCounter > 5 THEN
			b_MBComErrorActive := TRUE;
		END_IF
	END_IF
END_IF
END_METHOD

ACTION SFCTipReset:
SFCTip := FALSE;
END_ACTION

END_FUNCTION_BLOCK

(* stored: Version 1.1.0.1, ProductVersion 3.1.4026.18
   POU FB_BMS: Id {f84bc1e7-b567-4e5e-b38f-18427cbcc8bc}, SpecialFunc None
   Folder Internal methods: Id {65537688-ac4f-4f6d-b27a-a80fb821076a}
   Folder SFC: Id {564b7e00-10ec-45f5-9af8-1415fba4befa}
   Action aBMSPoweroff: Id {bc94f2c8-8a98-48e3-b5e9-e15077eca8d2}
   Action aBMSPowerOn: Id {b655e345-07db-4f12-84c2-cfe3522b2cf1}
   Action aClearFaults: Id {73544eea-c2c5-4fe8-9685-c28fe51514ac}
   Action aDisableInsulationMonitor: Id {b0c7eb78-8848-404e-b0c6-de98883fd0a5}
   Action aGetMBMUData: Id {9b9bbfba-6e9f-40a4-9614-b12703001d18}
   Action aGetSBMUData: Id {c2071653-1677-4e1e-b725-cb505e532c67}
   Action aGetStaticData: Id {4c3ada9c-4cf8-4cd8-b7cf-729c47af2d89}
   Action aGetStatus: Id {a90aa134-5027-48a9-8e91-d8356eeffd5b}
   Action aInit: Id {1bf09aae-72dd-46d8-8fb4-afdc9a2999c1}
   Action aSetDateTime: Id {f440fcdb-53bf-4a49-b2b3-caedac4d907e}
   Action aSetPowerMode: Id {c0cb5012-948e-4d4c-a5f7-7892e11c8df2}
   Action aWatchdog: Id {4862538b-5535-4b9c-8486-6240a5b4b5f4}
   Method BMS_Diagnostics: Id {e3c13309-b712-4d57-bb48-1ed0d35570ec}
   Method BMSDatalogger: Id {b558f9ed-5adf-4844-9721-435d0a77dafd}
   Method BMSHeartBeat: Id {fa0a650b-d9a2-4319-bbf8-8b86e69ebb7d}
   Action BMSSFC: Id {dccfe960-0abf-40f0-9ccc-feca3d4baf90}
   Method CalculateCumulativeValues: Id {3804fa2a-060f-428b-b8a6-7307214e863c}
   Method CalculatedRatings: Id {06d54167-e03f-47a0-9c1f-ca4905f9230b}
   Method CalculateSoCUser: Id {e6795d0b-c944-48b9-a172-f83a0022c355}
   Method CalculateTimeRemaining: Id {bfc8b221-1e23-4f03-a144-9954123c7e90}
   Method ClearBMSFaults: Id {5968c632-fac0-42cc-b87f-bb587cf9f857}
   Method EMSTOP: Id {2513f3ae-f229-4af9-b6f0-9384f5a93641}
   Method GetBatteryInfo: Id {c680a140-f52e-4b81-b2e8-bc3403eb77b3}
   Method GetCellData: Id {398e55a4-76bb-42bf-b2b2-e5c29576043c}
   Method GetDiagnostics: Id {4946c134-241c-4c4f-a711-8dcfd2dcc4b2}
   Method GetMBMUData: Id {2865fbe8-2bb0-4c3f-9529-febe10dc8e41}
   Method GetMBMUStaticSystemData: Id {a3301c10-905c-443a-9591-87c331836d2e}
   Method GetSBMUData: Id {87c82cc2-9d5a-42d1-9f20-3277e4813f1b}
   Method GetSBMUStaticSystemData: Id {83657047-15fc-4e44-a2cb-fc7cbd873b56}
   Method GetSystemStatus: Id {3238feeb-548c-429e-ba4f-29bd654b5254}
   Method GetWearCounters: Id {a4e51fcd-c5c4-40b1-9675-e15be5162629}
   Method Init: Id {0aceaa9b-4149-4430-9b55-09d9d046f8c9}
   Method OpenInsulationSwitch: Id {f96dd416-96e6-41c4-9643-9e191e336a6b}
   Method Reset: Id {7b3ba1ee-cf3d-4d9d-a084-997be89556e2}
   Method SetBMSDateTime: Id {9849d9aa-aeea-4099-8bb3-523b243ba620}
   Method SetPowerMode: Id {7f32a673-5053-4103-9dc6-69d9f8152fc9}
   Action SFCTipReset: Id {bd39e870-0e61-4d10-baf7-1dc4d7417da6} *)
